# B&R Automation Studio project AP124 (part 3)

#### conveyorP13P14Control.st - not listed in the package file held
```iecst
ACTION ConveyorP13P14Control:

	IF modePalletization = modePalletizationNotReadyToStart THEN
		stateConveyorP13P14 := stateConveyorStop;
	END_IF

	//detect pallet
	IF diPalletStopP14 THEN
		palletOnConveyorP14 := TRUE;
	END_IF

	CASE stateConveyorP13P14 OF

		stateConveyorStop:

			cmdMovePalletP13P14 := FALSE;
			doConveyorP13 := FALSE;
			acpI_P14.switchOn := TRUE;
			acpI_P14.speed := 0;
			acpI_P14.reset := TRUE;
			IF modePalletization <> modePalletizationNotReadyToStart THEN
				stateConveyorP13P14 := stateConveyorWait;
			END_IF

		stateConveyorWait:

			IF cmdMovePalletP13P14 THEN
				IF palletOnConveyorP14 AND NOT diReset THEN
					alarmImagePalletization[3] := TRUE;
					stateConveyorP12P13 := stateConveyorStop;
				ELSE
					TON_ConveyorP13P14(IN := FALSE);
					stateConveyorP13P14 := stateConveyorMoving;
				END_IF
			END_IF

			IF palletOnConveyorP14 > palletOnConveyorP14old THEN
				alarmImagePalletization[10] := TRUE;
				stateConveyorP13P14 := stateConveyorStop;
			END_IF

		stateConveyorMoving:

			doConveyorP13 := TRUE;
			acpI_P14.speed := 500;

			IF NOT cmdMovePalletP13P14 THEN
				stateConveyorP13P14 := stateConveyorStop;
			END_IF

			//sensor reached?
			IF diPalletSlowDownP14 THEN
				palletOnConveyorP13 := FALSE;
				TON_ConveyorP13P14(IN := FALSE);
				stateConveyorP13P14 := stateConveyorMovingSlow;
			END_IF

			//timeout?
			TON_ConveyorP13P14(IN := TRUE, PT := T#12s);
			IF TON_ConveyorP13P14.Q AND NOT diReset THEN
				alarmImagePalletization[4] := TRUE;
				stateConveyorP13P14 := stateConveyorStop;
			END_IF

		stateConveyorMovingSlow:

			acpI_P14.speed := 200;

			IF NOT cmdMovePalletP13P14 THEN
				stateConveyorP13P14 := stateConveyorStop;
			END_IF

			IF palletOnConveyorP14 AND NOT diReset THEN
				stateConveyorP13P14 := stateConveyorStop;
			END_IF

			//timeout?
			TON_ConveyorP13P14(IN := TRUE, PT := T#6s);
			IF TON_ConveyorP13P14.Q AND NOT diReset THEN
				alarmImagePalletization[2] := TRUE;
				stateConveyorP13P14 := stateConveyorStop;
			END_IF
	END_CASE

	//control of ACOPOSinverter P14
	acpI_P14();

	palletOnConveyorP14old := palletOnConveyorP14;

	alarmImagePalletization[13] := NOT diMotorProtectionP13;

	IF acknowledgeImagePalletization[2] THEN
		alarmImagePalletization[2] := FALSE;
	END_IF
	IF acknowledgeImagePalletization[3] THEN
		alarmImagePalletization[3] := FALSE;
	END_IF

	IF acknowledgeImagePalletization[4] THEN
		alarmImagePalletization[4] := FALSE;
	END_IF

	IF acknowledgeImagePalletization[10] THEN
		alarmImagePalletization[10] := FALSE;
	END_IF

	IF acpI_P14.error THEN
		alarmImagePalletization[24] := TRUE;
	ELSE
		alarmImagePalletization[24] := FALSE;
	END_IF

END_ACTION
```

#### conveyorP14.st - not listed in the package file held
```iecst
ACTION ConveyorP14:

	acpI_P14.switchOn := TRUE;
	acpI_P14.speed := 500;

	CASE statePalletP14 OF

		palletNotPresent:

			acpI_P14.run := (cmdMovePalletP14 AND (statePalletP15 = palletNotPresent OR diReset)) OR cmdMovePalletP13;

			//slow down sensor?
			IF diPalletSlowDownP14 THEN
				acpI_P14.speed := 200;
			END_IF

		palletPresent:

			IF cmdMovePalletP14 AND (statePalletP15 = palletNotPresent OR diReset) THEN
				statePalletP14 := palletMoving;
			END_IF

			acpI_P14.run := FALSE;

		palletMoving:

			//sensor reached?
			IF TON_PalletStopP15.Q AND cmdMovePalletP14 AND NOT diReset THEN
				statePalletP15 := palletPresent;
				statePalletP14 := palletNotPresent;
				cmdMovePalletP14 := FALSE;
			END_IF

			acpI_P14.run := cmdMovePalletP14;

	END_CASE

	//control of ACOPOSinverter
	acpI_P14();

END_ACTION
```

#### conveyorP14P15Control.st - not listed in the package file held
```iecst
ACTION ConveyorP14P15Control:

	IF modePalletization = modePalletizationNotReadyToStart THEN
		stateConveyorP14P15 := stateConveyorStop;
	END_IF

	//detect pallet
	IF diPalletStopP15 THEN
		palletOnConveyorP15 := TRUE;
	END_IF

	CASE stateConveyorP14P15 OF

		stateConveyorStop:

			cmdMovePalletP14P15 := FALSE;
			acpI_P14.switchOn := TRUE;
			acpI_P14.speed := 0;
			acpI_P14.reset := TRUE;
			acpI_P15.switchOn := TRUE;
			acpI_P15.speed := 0;
			acpI_P15.reset := TRUE;
			IF modePalletization <> modePalletizationNotReadyToStart THEN
				stateConveyorP14P15 := stateConveyorWait;
			END_IF

		stateConveyorWait:

			IF cmdMovePalletP14P15 THEN
				IF palletOnConveyorP15 AND NOT diReset THEN
					alarmImagePalletization[6] := TRUE;
					stateConveyorP14P15 := stateConveyorStop;
				ELSE
					TON_ConveyorP14P15(IN := FALSE);
					stateConveyorP14P15 := stateConveyorMoving;
				END_IF
			END_IF

			IF palletOnConveyorP15 > palletOnConveyorP15old THEN
				alarmImagePalletization[11] := TRUE;
				stateConveyorP14P15 := stateConveyorStop;
			END_IF

		stateConveyorMoving:

			acpI_P14.speed := 500;
			acpI_P15.speed := 500;

			IF NOT cmdMovePalletP14P15 THEN
				stateConveyorP14P15 := stateConveyorStop;
			END_IF

			//sensor reached?
			IF palletOnConveyorP15 AND NOT diReset THEN
				palletOnConveyorP14 := FALSE;
				stateConveyorP14P15 := stateConveyorStop;
			END_IF

			//timeout?
			TON_ConveyorP14P15(IN := TRUE, PT := T#12s);
			IF TON_ConveyorP14P15.Q AND NOT diReset THEN
				alarmImagePalletization[7] := TRUE;
				stateConveyorP14P15 := stateConveyorStop;
			END_IF

	END_CASE

	//control of ACOPOSinverter P15
	acpI_P15();

	palletOnConveyorP15old := palletOnConveyorP15;

	IF acknowledgeImagePalletization[6] THEN
		alarmImagePalletization[6] := FALSE;
	END_IF
	IF acknowledgeImagePalletization[7] THEN
		alarmImagePalletization[7] := FALSE;
	END_IF

	IF acknowledgeImagePalletization[11] THEN
		alarmImagePalletization[11] := FALSE;
	END_IF

	IF acpI_P15.error THEN
		alarmImagePalletization[25] := TRUE;
	ELSE
		alarmImagePalletization[25] := FALSE;
	END_IF

END_ACTION
```

#### conveyorP15.st - not listed in the package file held
```iecst
ACTION ConveyorP15:

	acpI_P15.switchOn := TRUE;
	acpI_P15.speed := 500;

	CASE statePalletP15 OF

		palletNotPresent:

			acpI_P15.run := (cmdMovePalletP15 AND (statePalletP16 = palletNotPresent OR diReset)) OR cmdMovePalletP14;

		palletPresent:

			IF cmdMovePalletP15 AND (statePalletP16 = palletNotPresent OR diReset) THEN
				statePalletP15 := palletMoving;
			END_IF

			acpI_P15.run := FALSE;

		palletMoving:

			//sensor reached?
			IF TON_PalletStopP16.Q AND cmdMovePalletP15 AND NOT diReset THEN
				statePalletP16 := palletPresent;
				statePalletP15 := palletNotPresent;
				cmdMovePalletP15 := FALSE;
			END_IF

			acpI_P15.run := cmdMovePalletP15;

	END_CASE

	//control of ACOPOSinverter
	acpI_P15();

END_ACTION
```

#### conveyorP16.st - not listed in the package file held
```iecst
ACTION ConveyorP16:

	acpI_P16.switchOn := TRUE;
	acpI_P16.speed := 500;

	CASE statePalletP16 OF

		palletNotPresent:

			acpI_P16.run := (cmdMovePalletP16 AND (statePalletP17 = palletNotPresent OR diReset)) OR cmdMovePalletP15;

		palletPresent:

			IF cmdMovePalletP16 AND (statePalletP17 = palletNotPresent OR diReset) THEN
				statePalletP16 := palletMoving;
			END_IF

			acpI_P16.run := FALSE;

		palletMoving:

			//sensor reached?
			IF TON_PalletStopP17.Q AND cmdMovePalletP16 AND NOT diReset THEN
				statePalletP17 := palletPresent;
				statePalletP16 := palletNotPresent;
				cmdMovePalletP16 := FALSE;
			END_IF

			acpI_P16.run := cmdMovePalletP16;

	END_CASE

	//control of ACOPOSinverter
	acpI_P16();

END_ACTION
```

#### conveyorP17.st - not listed in the package file held
```iecst
ACTION ConveyorP17:

	acpI_P17.switchOn := TRUE;
	acpI_P17.speed := 500;

	CASE statePalletP17 OF

		palletNotPresent:

			acpI_P17.run := (cmdMovePalletP17 AND (statePalletP18 = palletNotPresent OR diReset) AND stateTurnTable = stateTurnTableEntryPosition) OR cmdMovePalletP16;

		palletPresent:

			IF cmdMovePalletP17 AND (statePalletP18 = palletNotPresent OR diReset) THEN
				statePalletP17 := palletMoving;
			END_IF

			acpI_P17.run := FALSE;

		palletMoving:

			//sensor reached?
			IF TON_PalletStopP18.Q AND cmdMovePalletP17 AND NOT diReset THEN
				statePalletP18 := palletPresent;
				statePalletP17 := palletNotPresent;
				cmdMovePalletP17 := FALSE;
			END_IF

			acpI_P17.run := cmdMovePalletP17;

	END_CASE

	//control of ACOPOSinverter
	acpI_P17();

END_ACTION
```

### pallet_conveyors.typ - not listed in the package file held
```iecst
TYPE
	ModeConveyors :
		(
		modeConveyorsNotReadyToStart,
		modeConveyorsManual,
		modeConveyorsAuto
		);
END_TYPE
```

### outfeed.typ
```iecst
TYPE
	StateTurnTable :
		(
		stateTurnTableInit,
		stateTurnTableEntryPosition,
		stateTurnTableMovingToExitPos,
		stateTurnTableExitPosition,
		stateTurnTableMovingToEntryPos
		);
END_TYPE
```

### outfeed.var
```iecst
VAR
	acknowledgeImageOutfeed : ARRAY[0..39] OF BOOL;
	alarmImageOutfeed : ARRAY[0..39] OF BOOL;
	alarmInZoneOutfeed : BOOL;
	cmdMovePalletP17 : BOOL;
	cmdMovePalletP18 : BOOL;
	cmdOutfeedAuto : BOOL; (*VISU:switches pallet magazine to automatic mode*)
	cmdOutfeedManual : BOOL;
	diWrapperDoorCanBeOpened : BOOL;
	diWrapperEntryFree : BOOL;
	diWrapperExitFree : BOOL;
	diWrapperInAuto : BOOL;
	diWrapperLowFoil : BOOL;
	diWrapperNoError : BOOL;
	diWrappingFinished : BOOL;
	doWrapperNoExternalStop : BOOL;
	doWrapperSortiment1 : BOOL;
	doWrapperSortiment2 : BOOL;
	doWrappingStart : BOOL;
	modeZoneOutfeed : ModeZone;
	modeZoneOutfeedOld : ModeZone;
	statePalletP17 : StatePallet;
	statePalletP18 : StatePallet;
	statePalletP19 : StatePallet;
	statePalletP20 : StatePallet;
	statePalletP21 : StatePallet;
	statePalletP22 : StatePallet;
	stateTurnTable : StateTurnTable;
END_VAR
```

### Program Logical/plc/outfeed/outfeed_main (IEC) - palletization state machine

#### outfeed_main.st - Init, cyclic, exit code
```iecst
PROGRAM _INIT

END_PROGRAM

PROGRAM _CYCLIC

	modeZoneOutfeedOld := modeZoneOutfeed;

	readyToStart := NOT diOutfeedEDM;

	IF cpuIsSimulated THEN
		readyToStart := TRUE;
	END_IF

	IF NOT readyToStart THEN
		modeZoneOutfeed := modeZoneOff;
	END_IF

	CASE modeZoneOutfeed OF

		modeZoneOff: //the automat is not ready to start

			cmdOutfeedManual := FALSE;
			cmdOutfeedAuto := FALSE;

			IF readyToStart THEN
				modeZoneOutfeed := modeZoneManual;
			END_IF

		modeZoneManual:

			cmdOutfeedManual := FALSE;

			IF (NOT alarmInZoneOutfeed OR cpuIsSimulated) AND cmdOutfeedAuto THEN
				modeZoneOutfeed := modeZoneAuto;
			END_IF

		modeZoneAuto:

			cmdOutfeedAuto := FALSE;

			IF (alarmInZoneOutfeed AND NOT cpuIsSimulated) OR cmdOutfeedManual THEN
				modeZoneOutfeed := modeZoneManual;
			END_IF

	END_CASE

	//alarms
	alarmImageOutfeed[0] := NOT lightCurtainP17;
	alarmImageOutfeed[3] := NOT diMotorProtectionP19;
	alarmImageOutfeed[9] := NOT diMotorProtectionP20;
	alarmImageOutfeed[12] := NOT diMotorProtectionP21;
	alarmImageOutfeed[13] := NOT diMotorProtectionP22;
END_PROGRAM
```

#### outfeed_main.var - Local variables
```iecst
VAR
	readyToStart : BOOL;
	diMotorProtectionP19 : BOOL;
	diMotorProtectionP20 : BOOL;
	diMotorProtectionP21 : BOOL;
	diMotorProtectionP22 : BOOL;
	lightCurtainP17 : BOOL;
END_VAR
```

### Program Logical/plc/outfeed/pallet_outfeed/pallet_outfeed (IEC) - pallet outfeed control

#### Main.st - Cyclic code
```iecst
PROGRAM _INIT
	(* Insert code here *)

END_PROGRAM

PROGRAM _CYCLIC
	TON_PalletStopP18(IN := diPalletStopP18, PT := T#200ms);
	TON_PalletStopP20(IN := diPalletStopP20, PT := T#200ms);
	TON_PalletStopP21(IN := diPalletStopP21, PT := T#200ms);
	TON_PalletStopP22(IN := diPalletStopP22, PT := T#200ms);

	CASE modeZoneOutfeed OF

		modeZoneOff:

		modeZoneManual:

			IF modeZoneOutfeedOld <> modeZoneManual THEN
				cmdMovePalletP17 := FALSE;
				cmdMovePalletP19 := FALSE;
				cmdMovePalletP20 := FALSE;
				cmdMovePalletP21 := FALSE;
				cmdMovePalletP22 := FALSE;
			END_IF

		modeZoneAuto:

			//stop sensor not reached
			TON_ConveyorP17(IN := cmdMovePalletP17, PT := T#20s);
			alarmImageOutfeed[21] := TON_ConveyorP17.Q;

			TON_ConveyorP19(IN := cmdMovePalletP19, PT := T#20s);
			alarmImageOutfeed[1] := TON_ConveyorP19.Q;

			TON_ConveyorP20(IN := cmdMovePalletP20, PT := T#20s);
			alarmImageOutfeed[8] := TON_ConveyorP20.Q;

			TON_ConveyorP21(IN := cmdMovePalletP21, PT := T#20s);
			alarmImageOutfeed[11] := TON_ConveyorP21.Q;

			// control conveyors
			IF statePalletP17 <> palletNotPresent AND statePalletP18 = palletNotPresent AND stateTurnTable = stateTurnTableEntryPosition AND diWrapperEntryFree THEN
				cmdMovePalletP17 := TRUE;
			END_IF

			IF statePalletP19 <> palletNotPresent AND statePalletP20 = palletNotPresent THEN
				cmdMovePalletP19 := TRUE;
			END_IF

			IF statePalletP20 <> palletNotPresent AND statePalletP21 = palletNotPresent THEN
				cmdMovePalletP20 := TRUE;
			END_IF

			IF statePalletP21 <> palletNotPresent AND statePalletP22 = palletNotPresent THEN
				cmdMovePalletP21 := TRUE;
			END_IF

			//unexpected pallet
			IF TON_PalletStopP18.Q AND statePalletP18 = palletNotPresent AND NOT cmdMovePalletP17 AND stateTurnTable = stateTurnTableEntryPosition THEN
				alarmImageOutfeed[20] := TRUE;
			END_IF
			IF TON_PalletStopP20.Q AND statePalletP20 = palletNotPresent AND NOT cmdMovePalletP19 THEN
				alarmImageOutfeed[2] := TRUE;
			END_IF
			IF TON_PalletStopP21.Q AND statePalletP21 = palletNotPresent AND NOT cmdMovePalletP20 THEN
				alarmImageOutfeed[7] := TRUE;
			END_IF
			IF TON_PalletStopP22.Q AND statePalletP22 = palletNotPresent AND NOT cmdMovePalletP21 THEN
				alarmImageOutfeed[10] := TRUE;
			END_IF

	END_CASE

	//conveyors
	ConveyorP17;
	ConveyorP19;
	ConveyorP20;
	ConveyorP21;
	ConveyorP22;

	//stop sensor not reached
	IF acknowledgeImageOutfeed[21] THEN
		alarmImageOutfeed[21] := FALSE;
	END_IF
	IF acknowledgeImageOutfeed[1] THEN
		alarmImageOutfeed[1] := FALSE;
	END_IF
	IF acknowledgeImageOutfeed[8] THEN
		alarmImageOutfeed[8] := FALSE;
	END_IF
	IF acknowledgeImageOutfeed[11] THEN
		alarmImageOutfeed[11] := FALSE;
	END_IF

	//unexpected pallet
	IF acknowledgeImageOutfeed[20] THEN
		alarmImageOutfeed[20] := FALSE;
	END_IF
	IF acknowledgeImageOutfeed[2] THEN
		alarmImageOutfeed[2] := FALSE;
	END_IF
	IF acknowledgeImageOutfeed[7] THEN
		alarmImageOutfeed[7] := FALSE;
	END_IF
	IF acknowledgeImageOutfeed[10] THEN
		alarmImageOutfeed[10] := FALSE;
	END_IF

	//problems with motors
	acknowledgeImageOutfeed[22] := acpI_P17.error;
	acpI_P17.reset := EDGENEG(acknowledgeImageOutfeed[22]);

END_PROGRAM
```

#### Variables.var - Local variables
```iecst
VAR
	acpI_P17 : AcpInoSdc;
	cmdMovePalletP19 : BOOL;
	cmdMovePalletP20 : BOOL;
	cmdMovePalletP21 : BOOL;
	cmdMovePalletP22 : BOOL;
	diPalletStopP18 : BOOL;
	diPalletStopP20 : BOOL;
	diPalletStopP21 : BOOL;
	diPalletStopP22 : BOOL;
	doConveyorP19 : BOOL;
	doConveyorP20 : BOOL;
	doConveyorP21 : BOOL;
	doConveyorP22 : BOOL;
	TOF_PalletStopP22 : TOF;
	TON_ConveyorP17 : TON;
	TON_ConveyorP19 : TON;
	TON_ConveyorP20 : TON;
	TON_ConveyorP21 : TON;
	TON_PalletStopP18 : TON;
	TON_PalletStopP20 : TON;
	TON_PalletStopP21 : TON;
	TON_PalletStopP22 : TON;
END_VAR
```

#### conveyorP19.st
```iecst
ACTION ConveyorP19:

	CASE statePalletP19 OF

		palletNotPresent:

			doConveyorP19 := (cmdMovePalletP19 AND (statePalletP20 = palletNotPresent OR diReset)) OR (cmdMovePalletP18 AND stateTurnTable = stateTurnTableExitPosition);

		palletPresent:

			IF cmdMovePalletP19 AND (statePalletP20 = palletNotPresent OR diReset) THEN
				statePalletP19 := palletMoving;
			END_IF

			doConveyorP19 := FALSE;

		palletMoving:

			//sensor reached?
			IF TON_PalletStopP20.Q AND cmdMovePalletP19 AND NOT diReset THEN
				statePalletP20 := palletPresent;
				statePalletP19 := palletNotPresent;
				cmdMovePalletP19 := FALSE;
			END_IF

			doConveyorP19 := cmdMovePalletP19;

	END_CASE

END_ACTION
```

#### conveyorP20.st
```iecst
ACTION ConveyorP20:

	CASE statePalletP20 OF

		palletNotPresent:

			doConveyorP20 := (cmdMovePalletP20 AND (statePalletP21 = palletNotPresent OR diReset)) OR cmdMovePalletP19;

		palletPresent:

			IF cmdMovePalletP20 AND (statePalletP21 = palletNotPresent OR diReset) THEN
				statePalletP20 := palletMoving;
			END_IF

			doConveyorP20 := FALSE;

		palletMoving:

			//sensor reached?
			IF TON_PalletStopP21.Q AND cmdMovePalletP20 AND NOT diReset THEN
				statePalletP21 := palletPresent;
				statePalletP20 := palletNotPresent;
				cmdMovePalletP20 := FALSE;
			END_IF

			doConveyorP20 := cmdMovePalletP20;

	END_CASE

END_ACTION
```

#### conveyorP21.st
```iecst
ACTION ConveyorP21:

	CASE statePalletP21 OF

		palletNotPresent:

			doConveyorP21 := (cmdMovePalletP21 AND (statePalletP22 = palletNotPresent OR diReset)) OR cmdMovePalletP20;

		palletPresent:

			IF cmdMovePalletP21 AND (statePalletP22 = palletNotPresent OR diReset) THEN
				statePalletP21 := palletMoving;
			END_IF

			doConveyorP21 := FALSE;

		palletMoving:

			//sensor reached?
			IF TON_PalletStopP22.Q AND cmdMovePalletP21 AND NOT diReset THEN
				statePalletP22 := palletPresent;
				statePalletP21 := palletNotPresent;
				cmdMovePalletP21 := FALSE;
			END_IF

			doConveyorP21 := cmdMovePalletP21;

	END_CASE

END_ACTION
```

#### conveyorP22.st
```iecst
ACTION ConveyorP22:

	TOF_PalletStopP22(IN := diPalletStopP22, PT := T#30s);

	IF NOT TOF_PalletStopP22.Q THEN
		statePalletP22 := palletNotPresent;
	END_IF

	CASE statePalletP22 OF

		palletNotPresent:

			doConveyorP22 := (cmdMovePalletP22 AND diReset) OR cmdMovePalletP21;

		palletPresent:

			doConveyorP22 := FALSE;

		palletMoving:

			statePalletP22 := palletNotPresent;

	END_CASE

END_ACTION
```

### Program Logical/plc/outfeed/wrapper/wrapper (IEC)

#### Main.st - Cyclic code
```iecst
PROGRAM _INIT

	diWrapperDoorCanBeOpened;

END_PROGRAM

PROGRAM _CYCLIC

	IF adrRecipes = 0 THEN
		RETURN;
	END_IF

	dRecipes ACCESS adrRecipes;
	IF dRecipes.actualRecipeIndex < 0 OR dRecipes.actualRecipeIndex > 9 THEN
		RETURN;
	END_IF

	dActualRecipe ACCESS ADR(dRecipes.recipe[dRecipes.actualRecipeIndex]);

	doWrapperSortiment1 := dActualRecipe.wrapperSortiment.0;
	doWrapperSortiment2 := dActualRecipe.wrapperSortiment.1;

	IF testAtAtrima THEN
		diPalletStopP19 := FALSE;
	END_IF

	TON_PalletStopP19(IN := diPalletStopP19, PT := T#200ms);

	CASE modeZoneOutfeed OF

		modeZoneOff: //the automat is not ready to start

		modeZoneManual:

			IF modeZoneOutfeedOld <> modeZoneManual THEN
				cmdMovePalletP18 := FALSE;
			END_IF

			doWrapperNoExternalStop := TRUE;
			doWrappingStart := FALSE;
			stateAuto := stateAutoUndefined;

		modeZoneAuto:

			//stop sensor not reached
			TON_ConveyorP18(IN := cmdMovePalletP18, PT := T#20s);
			alarmImageOutfeed[4] := TON_ConveyorP18.Q;

			CASE stateAuto OF

				stateAutoUndefined:

					IF stateTurnTable = stateTurnTableEntryPosition THEN
						stateAuto := stateAutoWait;
					ELSE
						stateAuto := stateAutoRemovePallet;
					END_IF

				stateAutoWait:

					IF statePalletP18 = palletPresent AND stateTurnTable = stateTurnTableEntryPosition AND diWrapperInAuto THEN
						TON_Wrapper(IN:=FALSE);
						stateAuto := stateAutoWait2;
					END_IF

				stateAutoWait2:

					TON_Wrapper(IN:=TRUE, PT:=T#2s);
					IF TON_Wrapper.Q THEN
						stateAuto := stateAutoRun;
					END_IF

				stateAutoRun:

					doWrappingStart := TRUE;

					IF diWrappingFinished THEN
						stateAuto := stateAutoTurnToExitPosition;
					END_IF

				stateAutoTurnToExitPosition:

					doWrappingStart := FALSE;
					cmdTurnToExitPosition := TRUE;
					stateAuto := stateAutoWaitForExitPosition;

				stateAutoWaitForExitPosition:

					IF stateTurnTable = stateTurnTableExitPosition THEN
						stateAuto := stateAutoRemovePallet;
					END_IF

				stateAutoRemovePallet:

					IF statePalletP18 <> palletNotPresent AND statePalletP19 = palletNotPresent AND stateTurnTable = stateTurnTableExitPosition AND diWrapperExitFree THEN
						cmdMovePalletP18 := TRUE;
					END_IF

					IF statePalletP18 = palletNotPresent THEN
						stateAuto := stateAutoTurnToEntryPosition;
					END_IF

				stateAutoTurnToEntryPosition:

					cmdTurnToEntryPosition := TRUE;
					stateAuto := stateAutoWaitForEntryPosition;

				stateAutoWaitForEntryPosition:

					IF stateTurnTable = stateTurnTableEntryPosition THEN
						stateAuto := stateAutoWait;
					END_IF

			END_CASE

			//unexpected pallet
			IF TON_PalletStopP19.Q AND statePalletP19 = palletNotPresent AND NOT cmdMovePalletP18 THEN
				alarmImageOutfeed[5] := TRUE;
			END_IF
	END_CASE

	//modules
	ConveyorP18;
	TurnTable;

	//door logic
	DoorLogic_2();
	alarmImageOutfeed[15] := NOT DoorLogic_2.diDoorLocked;

	alarmImageOutfeed[16] := wrapperEdmError;
	alarmImageOutfeed[17] := NOT diWrapperNoError;
	alarmImageOutfeed[18] := diWrapperLowFoil;
	alarmImageOutfeed[19] := NOT diWrapperInAuto;

	//sensor not reached
	IF acknowledgeImageOutfeed[4] THEN
		alarmImageOutfeed[4] := FALSE;
	END_IF

	//unexpected pallet
	IF acknowledgeImageOutfeed[5] THEN
		alarmImageOutfeed[5] := FALSE;
	END_IF

	//problems with motors
	alarmImageOutfeed[6] := acpI_P18_1.error;
	acpI_P18_1.reset := EDGENEG(acknowledgeImageOutfeed[6]);

	alarmImageOutfeed[14] := acpI_P18_2.error;
	acpI_P18_2.reset := EDGENEG(acknowledgeImageOutfeed[14]);

END_PROGRAM
```

#### Types.typ - Local data types
```iecst
TYPE
	StateAuto :
		(
		stateAutoUndefined,
		stateAutoWait,
		stateAutoWait2,
		stateAutoRun,
		stateAutoTurnToExitPosition,
		stateAutoWaitForExitPosition,
		stateAutoRemovePallet,
		stateAutoTurnToEntryPosition,
		stateAutoWaitForEntryPosition
		);
END_TYPE
```

#### Variables.var - Local variables
```iecst
VAR
	acpI_P18_1 : AcpInoSdc;
	acpI_P18_2 : AcpInoSdc;
	cmdTurnToEntryPosition : BOOL;
	cmdTurnToExitPosition : BOOL;
	conveyorP18speed : INT;
	diEntrySwitch : BOOL;
	diExitSwitch : BOOL;
	diPalletStopP19 : BOOL;
	DoorLogic_2 : DoorLogic;
	TON_ConveyorP18 : TON;
	TON_PalletStopP19 : TON;
	turnTableSpeed : INT;
	wrapperEdmError : BOOL;
	stateAuto : StateAuto;
	dRecipes : REFERENCE TO Recipes;
	dActualRecipe : REFERENCE TO Recipe;
	TON_Wrapper : TON;
END_VAR
```

#### conveyorP18.st
```iecst
ACTION ConveyorP18:

	acpI_P18_1.switchOn := TRUE;
	conveyorP18speed := 635;//500;

	IF stateTurnTable = stateTurnTableEntryPosition THEN
		acpI_P18_1.speed := conveyorP18speed;
	END_IF

	IF stateTurnTable = stateTurnTableExitPosition THEN
		acpI_P18_1.speed := -conveyorP18speed;
	END_IF

	CASE statePalletP18 OF

		palletNotPresent:

			acpI_P18_1.run := (cmdMovePalletP18 AND (statePalletP18 = palletNotPresent OR diReset)) OR (cmdMovePalletP17 AND stateTurnTable = stateTurnTableEntryPosition);

		palletPresent:

			IF cmdMovePalletP18 AND (statePalletP19 = palletNotPresent OR diReset) THEN
				statePalletP18 := palletMoving;
			END_IF

			acpI_P18_1.run := FALSE;

		palletMoving:

			//sensor reached?
			IF TON_PalletStopP19.Q AND cmdMovePalletP18 AND NOT diReset THEN
				statePalletP19 := palletPresent;
				statePalletP18 := palletNotPresent;
				cmdMovePalletP18 := FALSE;
			END_IF

			acpI_P18_1.run := cmdMovePalletP18 AND (stateTurnTable = stateTurnTableExitPosition);

	END_CASE

	//lock movement
	IF stateTurnTable <> stateTurnTableEntryPosition AND stateTurnTable <> stateTurnTableExitPosition THEN
		acpI_P18_1.run := FALSE;
	END_IF

	//control of ACOPOSinverter
	acpI_P18_1();

END_ACTION
```

#### turnTable.st
```iecst
ACTION TurnTable:

	acpI_P18_2.switchOn := TRUE;
	turnTableSpeed := 1500;

	CASE stateTurnTable OF

		stateTurnTableInit:

			acpI_P18_2.run := FALSE;

			IF diEntrySwitch THEN
				stateTurnTable := stateTurnTableEntryPosition;
			END_IF

			IF diExitSwitch THEN
				stateTurnTable := stateTurnTableExitPosition;
			END_IF

			IF stateTurnTable = stateTurnTableInit THEN

				IF cmdTurnToEntryPosition THEN
					stateTurnTable := stateTurnTableMovingToEntryPos;
				END_IF

				IF cmdTurnToExitPosition THEN
					stateTurnTable := stateTurnTableMovingToExitPos;
				END_IF
			END_IF

		stateTurnTableEntryPosition:

			IF cmdTurnToExitPosition THEN
				stateTurnTable := stateTurnTableMovingToExitPos;
			END_IF

			cmdTurnToEntryPosition := FALSE;

		stateTurnTableMovingToExitPos:

			acpI_P18_2.speed := turnTableSpeed;
			acpI_P18_2.run := TRUE;

			IF diExitSwitch OR NOT cmdTurnToExitPosition THEN
				StopMovement;
			END_IF

		stateTurnTableExitPosition:

			IF cmdTurnToEntryPosition THEN
				stateTurnTable := stateTurnTableMovingToEntryPos;
			END_IF

			cmdTurnToExitPosition := FALSE;

		stateTurnTableMovingToEntryPos:

			acpI_P18_2.speed := -turnTableSpeed;
			acpI_P18_2.run := TRUE;

			IF diEntrySwitch OR NOT cmdTurnToEntryPosition THEN
				StopMovement;
			END_IF

	END_CASE

	//control of ACOPOSinverter
	acpI_P18_2();

END_ACTION

ACTION StopMovement:
	cmdTurnToEntryPosition := FALSE;
	cmdTurnToExitPosition := FALSE;
	stateTurnTable := stateTurnTableInit;
END_ACTION
```

### alarm_management.var
```iecst
VAR
	alarmCommon : BOOL;
	alarmImageCommon : ARRAY[0..39] OF BOOL;
	alarmInZoneMagazine : BOOL; (*VISU:there is at least one alarm in pallet magazine*)
	cpuIsSimulated : BOOL;
	diAirPresureOK : BOOL; (*VISU: 1...air pressure OK*)
	diReset : BOOL; (*acknowledges all errors*)
	alarmPresent : BOOL;
	safetyAlive : BOOL;
END_VAR
```

### Program Logical/plc/alarm_management/alarm_management (IEC) - alarm management

#### Variables.var
```iecst
VAR
	acknowledgeImage : ARRAY[0..39] OF BOOL;
	diEStop1 : BOOL; (*emergency stop 1*)
	diEStop2 : BOOL; (*emergency stop 2*)
	diEStop3 : BOOL; (*emergency stop 3*)
	diEStop4 : BOOL; (*emergency stop 4*)
	diEStopRobot : BOOL; (*emergency stop - robot*)
	diEStopWrapper : BOOL; (*emergency stop wrapper*)
	i : INT;
	magazineEdmError : BOOL; (*1=power on*)
	outfeedEdmError : BOOL; (*1=power on*)
	palletizationEdmError : BOOL; (*1=power on*)
	diEStop5 : BOOL;
END_VAR
```

#### Cyclic.st
```iecst
PROGRAM _CYCLIC

	MpAlarmXCore_0.MpLink := ADR(gAlarmXCore);
	MpAlarmXCore_0.Enable := 1;

	MpAlarmXCore_0();

	MpAlarmXListUI_0.MpLink := ADR(gAlarmXCore);
	MpAlarmXListUI_0.Enable := 1;
	MpAlarmXListUI_0.UIConnect := ADR(MpAlarmXListUIConnect);
	MpAlarmXListUI_0();

	IF diAirPresureOK THEN
		MpAlarmXReset(gAlarmXCore,'AirPressureNotOK');
	ELSE
		MpAlarmXSet(gAlarmXCore,'AirPressureNotOK');
	END_IF

	IF EDGEPOS(diReset) THEN
		MpAlarmXListUIConnect.AcknowledgeAll := TRUE;
	END_IF

END_PROGRAM
```

#### Main.st
```iecst
PROGRAM _INIT

	cpuIsSimulated := DiagCpuIsSimulated();

END_PROGRAM

PROGRAM _CYCLIC

	alarmImageCommon[0] := NOT diAirPresureOK;
	alarmImageCommon[1] := NOT diEStop1;
	alarmImageCommon[2] := NOT diEStop2;
	alarmImageCommon[3] := NOT diEStop3;
	alarmImageCommon[4] := NOT diEStop4;
	alarmImageCommon[14] := NOT diEStop5;

	alarmImageCommon[5] := NOT diEStopRobot;
	alarmImageCommon[6] := NOT diEStopWrapper;
	alarmImageCommon[7] := NOT safetyAlive;

	alarmImageCommon[8] := diMagazineEDM;
	alarmImageCommon[9] := diPalletizationEDM;
	alarmImageCommon[10] := diOutfeedEDM;
	alarmImageCommon[11] := magazineEdmError;
	alarmImageCommon[12] := palletizationEdmError;
	alarmImageCommon[13] := outfeedEdmError;

	//detect if there is any alarm
	alarmCommon := FALSE;
	FOR i:=0 TO 39 DO
		IF alarmImageCommon[i] OR acknowledgeImage[i] THEN
			alarmCommon := TRUE;
		END_IF
	END_FOR

	//detect if there is any alarm in zone Magazine
	alarmInZoneMagazine := FALSE;
	FOR i:=0 TO 39 DO
		IF alarmImageMagazine[i] OR acknowledgeImageMagazine[i] THEN
			alarmInZoneMagazine := TRUE;
		END_IF
	END_FOR

	//detect if there is any alarm in zone Palletization
	alarmInZonePalletization := FALSE;
	FOR i:=0 TO 69 DO
		IF alarmImagePalletization[i] OR acknowledgeImagePalletization[i] THEN
			alarmInZonePalletization := TRUE;
		END_IF
	END_FOR

	//detect if there is any alarm in zone Outfeed
	alarmInZoneOutfeed := FALSE;
	FOR i:=0 TO 39 DO
		IF alarmImageOutfeed[i] OR acknowledgeImageOutfeed[i] THEN
			alarmInZoneOutfeed := TRUE;
		END_IF
	END_FOR

	IF alarmCommon OR alarmInZoneMagazine OR alarmInZonePalletization OR alarmInZoneOutfeed THEN
		alarmPresent := TRUE;
	ELSE
		alarmPresent := FALSE;
	END_IF

END_PROGRAM
```

### recipe_management.typ
```iecst
TYPE
	Layout : 	STRUCT
		nbOfTrays : INT;
		tray : ARRAY[0..39]OF Tray;
	END_STRUCT;
	Recipe : 	STRUCT
		name : STRING[80];
		interlayerSheetBottom : BOOL;
		interlayerSheetTop : BOOL;
		conveyorP1speed : INT;
		conveyorP2speed : INT;
		timeAfterLastTrayInRow : TIME;
		timeDelayForTurn : TIME;
		nbOfLayers : INT;
		layer : ARRAY[0..9]OF INT;
	END_STRUCT;
	Recipes : 	STRUCT
		actualRecipeIndex : INT;
		recipe : ARRAY[0..9]OF Recipe;
		layout : ARRAY[0..9]OF Layout;
	END_STRUCT;
	Tray : 	STRUCT
		turnTray : BOOL;
		lastTray : LastTray;
	END_STRUCT;
	LastTray :
		(
		lastTrayNo,
		lastTrayInRow,
		lastTrayInHalfLayer,
		lastTrayInLayer
		);
END_TYPE
```

### recipe_management.var
```iecst
VAR
	adrRecipes : UDINT;
END_VAR
```

### Program Logical/plc/recipe_management/recipe_management (IEC)

#### Types.typ
```iecst
TYPE
	StateRecipe :
		(
		stateRecipeError,
		stateRecipeInit,
		stateRecipeWait,
		stateRecipeLoad,
		stateRecipeLoad2,
		stateRecipeLoad3,
		stateRecipeSave,
		stateRecipeSave2,
		stateRecipeSave3
		);
END_TYPE
```

#### Variables.var
```iecst
VAR
	cmdLoad : BOOL;
	cmdSave : BOOL;
	MpRecipeCsv_0 : MpRecipeCsv;
	MpRecipeRegPar_0 : MpRecipeRegPar;
	readyToStart : BOOL;
	recipes : Recipes;
	stateRecipe : StateRecipe;
END_VAR
```

#### Main.st
```iecst
PROGRAM _INIT

END_PROGRAM

PROGRAM _CYCLIC

	adrRecipes := ADR(recipes);

	readyToStart :=  NOT MpRecipeRegPar_0.Error AND NOT MpRecipeCsv_0.Error;

	IF NOT readyToStart THEN
		stateRecipe := stateRecipeError;
	END_IF

	CASE stateRecipe OF

		stateRecipeError:

			cmdLoad := FALSE;
			cmdSave := FALSE;
			VisuRecipeState := 4;							//Visu Error Text
			IF readyToStart THEN
				stateRecipe := stateRecipeInit;
			END_IF

		stateRecipeInit:

			MpRecipeRegPar_0.MpLink := ADR(gRecipeCsv);
			MpRecipeRegPar_0.Enable := TRUE;
			MpRecipeRegPar_0.PVName := ADR('recipe_man:recipes');

			MpRecipeCsv_0.MpLink := ADR(gRecipeCsv);
			MpRecipeCsv_0.Enable := TRUE;
			MpRecipeCsv_0.DeviceName := ADR('USER');
			MpRecipeCsv_0.FileName := ADR('recipe.csv');

			VisuRecipeState := 0;						//Visu Empty Text

			IF MpRecipeRegPar_0.Active AND MpRecipeCsv_0.Active THEN
				stateRecipe := stateRecipeLoad;
			END_IF

		stateRecipeWait:

			IF cmdLoad THEN
				stateRecipe := stateRecipeLoad;
			END_IF

			IF cmdSave THEN
				stateRecipe := stateRecipeSave;
			END_IF

		stateRecipeLoad:

			MpRecipeCsv_0.Load := TRUE;
			stateRecipe := stateRecipeLoad2;
			VisuRecipeState := 3;						//Visu Discart changes Text

		stateRecipeLoad2:

			IF MpRecipeCsv_0.CommandDone THEN
				cmdLoad := FALSE;
				MpRecipeCsv_0.Load := FALSE;
				stateRecipe := stateRecipeWait;
				VisuRecipeState := 0;					//Visu Empty Text
				RecipeChanged := TRUE;
			END_IF

		stateRecipeSave:

			MpRecipeCsv_0.Save := TRUE;
			stateRecipe := stateRecipeSave2;
			VisuRecipeState := 1;						//Visu Saving Text

		stateRecipeSave2:

			IF MpRecipeCsv_0.CommandDone THEN
				cmdSave := FALSE;
				MpRecipeCsv_0.Save := FALSE;
				stateRecipe := stateRecipeWait;
				VisuRecipeState := 2;					//Visu Saved Text
				RecipeChanged := TRUE;
			END_IF

	END_CASE

	MpRecipeRegPar_0();
	MpRecipeCsv_0();

END_PROGRAM

PROGRAM _EXIT
	MpRecipeRegPar_0(Enable := FALSE);
	MpRecipeCsv_0(Enable := FALSE);
END_PROGRAM
```

### misc.var
```iecst
VAR
	testAtAtrima : BOOL;
	diActivateAllSafetyCircuits : BOOL; (*button on main cabinet to activate all safety circuits*)
	diMagazineEDM : BOOL; (*magazine safety zone: 0...contactor switched on*)
	diPalletizationEDM : BOOL; (*paletization safety zone: 0...contactor switched on*)
	diOutfeedEDM : BOOL; (*wrapper+outfeed safety zone: 0...contactor switched on*)
END_VAR
```

### Program Logical/plc/misc/misc

#### Variables.var
```iecst
VAR
	doLedOn : BOOL; (*LED indicator on main cabinet*)
	doLedOff : BOOL; (*LED indicator on main cabinet*)
	MTBasicsPWM_2 : MTBasicsPWM;
	MTBasicsPWM_1 : MTBasicsPWM;
	MTBasicsPWM_0 : MTBasicsPWM;
	sumEDM : INT;
	doSafetyCurtainSupplyP15 : BOOL;
	doSafetyCurtainSupplyP17 : BOOL;
	doSafetyCurtainSupplyP11 : BOOL;
	doSignColumnGreen : BOOL;
	doSignColumnOrange : BOOL;
	doSignColumnRed : BOOL;
	doSignColumnHorn : BOOL;
	sumAuto : INT;
	bypassHorn : BOOL;
END_VAR
```

#### Main.st
```iecst
PROGRAM _INIT

	doSafetyCurtainSupplyP11 := TRUE;
	doSafetyCurtainSupplyP15 := TRUE;
	doSafetyCurtainSupplyP17 := TRUE;

END_PROGRAM

PROGRAM _CYCLIC

	sumEDM := BOOL_TO_INT(diMagazineEDM) + BOOL_TO_INT(diPalletizationEDM) + BOOL_TO_INT(diOutfeedEDM);

	CASE sumEDM OF
		0:
			MTBasicsPWM_0.DutyCycle := 100;
		1:
			MTBasicsPWM_0.DutyCycle := 50;
		2:
			MTBasicsPWM_0.DutyCycle := 50;
		3:
			MTBasicsPWM_0.DutyCycle := 0;
	END_CASE

	MTBasicsPWM_0(Enable := 1, Period := 1);

	doLedOn := MTBasicsPWM_0.Out AND safetyAlive;

	doLedOff := NOT doLedOn;

	diActivateAllSafetyCircuits;

	//signalization column
	doSignColumnRed := doLedOff;

	sumAuto := BOOL_TO_INT(modeZoneMagazine = modeZoneAuto) + BOOL_TO_INT(modeZonePalletization = modeZoneAuto) + BOOL_TO_INT(modeZoneOutfeed = modeZoneAuto);

	CASE sumAuto OF
		0:
			MTBasicsPWM_1.DutyCycle := 0;
		1:
			MTBasicsPWM_1.DutyCycle := 50;
		2:
			MTBasicsPWM_1.DutyCycle := 50;
		3:
			MTBasicsPWM_1.DutyCycle := 100;
	END_CASE

	MTBasicsPWM_1(Enable := 1, Period := 1);

	doSignColumnGreen := MTBasicsPWM_1.Out;

	//horn
	MTBasicsPWM_2(Enable := alarmPresent OR magazineEmpty OR interlayerSheetMagazineEmpty, DutyCycle := 50, Period := 1);

	doSignColumnOrange := MTBasicsPWM_2.Out OR bypassHorn;

	doSignColumnHorn := MTBasicsPWM_2.Out AND NOT bypassHorn;

	IF testAtAtrima THEN
		doSignColumnHorn := FALSE;
	END_IF

	IF NOT alarmPresent THEN
		bypassHorn := FALSE;
	END_IF

	IF alarmPresent AND diReset THEN
		bypassHorn := TRUE;
	END_IF

END_PROGRAM
```

### pallet_conveyors.var
```iecst
VAR
	modeConveyors : ModeConveyors;
	palletOnConveyorP13 : BOOL; (*VISU:pallet lies on conveyor*)
	palletOnConveyorP14 : BOOL;
	palletOnConveyorP15 : BOOL;
END_VAR
```

### Program Logical/plc/pallet_conveyors/pallet_conveyors (IEC) - pallet conveyors control

#### Main.st - Cyclic code
```iecst
PROGRAM _INIT
	(* Insert code here *)

END_PROGRAM

PROGRAM _CYCLIC

	readyToStart := NOT diPalletizationEDM;

	IF NOT readyToStart THEN
		modeConveyors := modeConveyorsNotReadyToStart;
	END_IF

	CASE modeConveyors OF

		modeConveyorsNotReadyToStart: //the automat is not ready to start

			IF readyToStart THEN
				modeConveyors := modeConveyorsManual;
			END_IF

		modeConveyorsManual:

			IF NOT alarmInZoneConveyors AND cmdAuto THEN
				cmdAuto := FALSE;
				modeConveyors := modeConveyorsAuto;
			END_IF
			cmdManual := FALSE;

		modeConveyorsAuto:

			IF alarmInZoneConveyors OR cmdManual THEN
				modeConveyors := modeConveyorsManual;
			END_IF

			IF palletOnConveyorP12 AND NOT palletOnConveyorP13 THEN
				cmdMovePalletP12P13 := TRUE;
			END_IF

			IF palletOnConveyorP13 AND NOT palletOnConveyorP14 THEN
				cmdMovePalletP13P14 := TRUE;
			END_IF

			IF palletOnConveyorP14 AND NOT palletOnConveyorP15 THEN
				cmdMovePalletP14P15 := TRUE;
			END_IF

	END_CASE

	//conveyor P12 + P13
	ConveyorP12P13Control;
	ConveyorP13P14Control;
	ConveyorP14P15Control;

	alarmImage[5] := NOT lightCurtainP15;
	alarmImage[8] := NOT lightCurtainP17;

	//detect if there is any alarm
	alarmInZoneConveyors := FALSE;
	FOR i:=0 TO 39 DO
		IF alarmImage[i] OR acknowledgeImage[i] THEN
			alarmInZoneConveyors := TRUE;
		END_IF
	END_FOR

END_PROGRAM
```

#### Types.typ - Local data types
```iecst
TYPE
	StateAuto :
		(
		stateAutoUndefined,
		stateAutoWaitForPallet,
		stateAutoMovePallet,
		stateAutoWaitForSensor
		);
	StateConveyor :
		(
		stateConveyorStop,
		stateConveyorWait,
		stateConveyorMoving
		);
END_TYPE
```

#### Variables.var - Local variables
```iecst
VAR
	acknowledgeImage : ARRAY[0..39] OF BOOL;
	acpI_P14 : AcpInoSdc;
	acpI_P15 : AcpInoSdc;
	alarmImage : ARRAY[0..39] OF BOOL;
	alarmInZoneConveyors : BOOL;
	cmdAuto : BOOL; (*VISU:switches pallet magazine to automatic mode*)
	cmdManual : BOOL;
	cmdMovePalletP12P13 : BOOL;
	cmdMovePalletP13P14 : BOOL;
	cmdMovePalletP14P15 : BOOL;
	diPalletSlowDownP14 : BOOL;
	diPalletStopP13 : BOOL;
	diPalletStopP14 : BOOL;
	diPalletStopP15 : BOOL;
	doConveyorP12 : BOOL; (*starts conveyor P12*)
	doConveyorP13 : BOOL;
	i : INT;
	lightCurtainP15 : BOOL;
	readyToStart : BOOL;
	stateConveyorP12P13 : StateConveyor;
	stateConveyorP13P14 : StateConveyor;
	stateConveyorP14P15 : StateConveyor;
	TON_ConveyorP12P13 : TON;
	TON_ConveyorP13P14 : TON;
	TON_ConveyorP14P15 : TON;
END_VAR
```

#### conveyorP12P13Control.st
```iecst
ACTION ConveyorP12P13Control:

	IF modeMagazine = modeMagazineNotReadyToStart THEN
		stateConveyorP12P13 := stateConveyorStop;
	END_IF

	CASE stateConveyorP12P13 OF

		stateConveyorStop:

			cmdMovePalletP12P13 := FALSE;
			doConveyorP12 := FALSE;
			doConveyorP13 := FALSE;
			stateConveyorP12P13 := stateConveyorWait;

		stateConveyorWait:

			IF cmdMovePalletP12P13 THEN
				IF palletOnConveyorP13 THEN
					alarmImage[1] := TRUE;
					stateConveyorP12P13 := stateConveyorStop;
				ELSE
					TON_ConveyorP12P13(IN := FALSE);
					stateConveyorP12P13 := stateConveyorMoving;
				END_IF
			END_IF

		stateConveyorMoving:

			doConveyorP12 := TRUE;
			doConveyorP13 := TRUE;

			//start timer
			TON_ConveyorP12P13(IN := TRUE, PT := T#12s);

			IF NOT cmdMovePalletP12P13 THEN
				stateConveyorP12P13 := stateConveyorStop;
			END_IF

			//sensor reached?
			IF palletOnConveyorP13 THEN
				palletOnConveyorP12 := FALSE;
				stateConveyorP12P13 := stateConveyorStop;
			END_IF

			//timeout?
			IF TON_ConveyorP12P13.Q THEN
				alarmImage[0] := TRUE;
				stateConveyorP12P13 := stateConveyorStop;
			END_IF

	END_CASE

	//detect pallet on conveyor
	IF diPalletStopP13 THEN
		palletOnConveyorP13 := TRUE;
	END_IF

	//edge alarms
	IF acknowledgeImage[0] THEN
		alarmImage[0] := FALSE;
	END_IF
	IF acknowledgeImage[1] THEN
		alarmImage[1] := FALSE;
	END_IF
END_ACTION
```

#### conveyorP13P14Control.st
```iecst
ACTION ConveyorP13P14Control:

	IF modeConveyors = modeConveyorsNotReadyToStart THEN
		stateConveyorP13P14 := stateConveyorStop;
	END_IF

	CASE stateConveyorP13P14 OF

		stateConveyorStop:

			cmdMovePalletP13P14 := FALSE;
			doConveyorP13 := FALSE;
			acpI_P14.switchOn := TRUE;
			acpI_P14.speed := 0;
			acpI_P14.reset := TRUE;
			stateConveyorP13P14 := stateConveyorWait;

		stateConveyorWait:

			IF cmdMovePalletP13P14 THEN
				IF palletOnConveyorP14 THEN
					alarmImage[3] := TRUE;
					stateConveyorP12P13 := stateConveyorStop;
				ELSE
					TON_ConveyorP13P14(IN := FALSE);
					stateConveyorP13P14 := stateConveyorMoving;
				END_IF
			END_IF

		stateConveyorMoving:

			doConveyorP13 := TRUE;
			acpI_P14.speed := 500;

			IF NOT cmdMovePalletP13P14 THEN
				stateConveyorP13P14 := stateConveyorStop;
			END_IF

			//sensor reached?
			IF diPalletSlowDownP14 THEN
				palletOnConveyorP13 := FALSE;
				TON_ConveyorP13P14(IN := FALSE);
				stateConveyorP13P14 := stateConveyorMovingSlow;
			END_IF

			//timeout?
			TON_ConveyorP13P14(IN := TRUE, PT := T#12s);
			IF TON_ConveyorP13P14.Q THEN
				alarmImage[4] := TRUE;
				stateConveyorP13P14 := stateConveyorStop;
			END_IF

		stateConveyorMovingSlow:

			acpI_P14.speed := 200;

			IF NOT cmdMovePalletP13P14 THEN
				stateConveyorP13P14 := stateConveyorStop;
			END_IF

			IF diPalletStopP14 THEN
				stateConveyorP13P14 := stateConveyorStop;
			END_IF

			//timeout?
			TON_ConveyorP13P14(IN := TRUE, PT := T#6s);
			IF TON_ConveyorP13P14.Q THEN
				alarmImage[2] := TRUE;
				stateConveyorP13P14 := stateConveyorStop;
			END_IF
	END_CASE

	//control of ACOPOSinverter P14
	acpI_P14();

	//detect pallet
	IF diPalletStopP14 THEN
		palletOnConveyorP14 := TRUE;
	END_IF

	//edge alarms
	IF acknowledgeImage[2] THEN
		alarmImage[2] := FALSE;
	END_IF
	IF acknowledgeImage[3] THEN
		alarmImage[3] := FALSE;
	END_IF
	IF acknowledgeImage[4] THEN
		alarmImage[4] := FALSE;
	END_IF

END_ACTION
```

#### conveyorP13Control.st - not listed in the package file held
```iecst
ACTION ConveyorP13Control:

	//detect pallet on conveyor
	IF diPalletOnConveyorP13 THEN
		palletOnConveyorP13 := TRUE;
	END_IF

END_ACTION
```

#### conveyorP14P15Control.st - not listed in the package file held
```iecst
ACTION ConveyorP14P15Control:

	IF modeConveyors = modeConveyorsNotReadyToStart THEN
		stateConveyorP14P15 := stateConveyorStop;
	END_IF

	CASE stateConveyorP14P15 OF

		stateConveyorStop:

			cmdMovePalletP14P15 := FALSE;
			acpI_P14.switchOn := TRUE;
			acpI_P14.speed := 0;
			acpI_P14.reset := TRUE;
			acpI_P15.switchOn := TRUE;
			acpI_P15.speed := 0;
			acpI_P15.reset := TRUE;
			stateConveyorP14P15 := stateConveyorWait;

		stateConveyorWait:

			IF cmdMovePalletP14P15 THEN
				IF palletOnConveyorP15 THEN
					alarmImage[6] := TRUE;
					stateConveyorP14P15 := stateConveyorStop;
				ELSE
					TON_ConveyorP14P15(IN := FALSE);
					stateConveyorP14P15 := stateConveyorMoving;
				END_IF
			END_IF

		stateConveyorMoving:

			acpI_P14.speed := 500;
			acpI_P15.speed := 500;

			IF NOT cmdMovePalletP14P15 THEN
				stateConveyorP14P15 := stateConveyorStop;
			END_IF

			//sensor reached?
			IF diPalletStopP15 THEN
				palletOnConveyorP14 := FALSE;
				stateConveyorP14P15 := stateConveyorStop;
			END_IF

			//timeout?
			TON_ConveyorP14P15(IN := TRUE, PT := T#12s);
			IF TON_ConveyorP14P15.Q THEN
				alarmImage[7] := TRUE;
				stateConveyorP14P15 := stateConveyorStop;
			END_IF

	END_CASE

	//control of ACOPOSinverter P15
	acpI_P15();

	//detect pallet
	IF diPalletStopP15 THEN
		palletOnConveyorP15 := TRUE;
	END_IF

	//edge alarms
	IF acknowledgeImage[6] THEN
		alarmImage[6] := FALSE;
	END_IF
	IF acknowledgeImage[7] THEN
		alarmImage[7] := FALSE;
	END_IF

END_ACTION
```

### pallet_outfeed.var
```iecst
VAR
	statusMessageOutfeed : INT;
END_VAR
```

### Program Logical/plc/pallet_outfeed/pallet_outfeed/pallet_outfeed

#### Main.st
```iecst
PROGRAM _INIT
	(* Insert code here *)

END_PROGRAM

PROGRAM _CYCLIC
	statusMessageOutfeed;

END_PROGRAM
```

### Program Logical/plc/pallet_outfeed/wrapper/wrapper (IEC) - wrapper control

#### Variables.var
```iecst
VAR
	diDoor2opened : BOOL;
	diOpenDoors2 : BOOL; (*button to open doors*)
	diCloseDoors2 : BOOL; (*button to close doors*)
END_VAR
```

### Program Logical/plc/pallett_magazine/pallet_magazine

#### Variables.var
```iecst
VAR
	armsState : ArmsState; (*VISU:arms state*)
	closeArms : BOOL; (*valve to close the arms*)
	cmdAutomatMode : BOOL; (*3 funkce v 1 (reset safety+ovladaci obvody + start automatu)*)
	cmdCloseArms : BOOL; (*VISU:command to close the arms*)
	cmdManualMode : BOOL; (*VISU:switches pallet magazine to manual mode*)
	cmdDown : BOOL; (*VISU:go with magazine up*)
	cmdUp : BOOL; (*VISU:go with magazine down*)
	moveToLowerPosition : BOOL; (*go with magazine to lower position*)
	moveToMiddlePosition : BOOL; (*go with magazine to middle position*)
	moveToUpperPosition : BOOL; (*go with magazine to upper position*)
	cmdOpenArms : BOOL; (*VISU:commad to open the arms*)
	leftArmClosed : BOOL; (*left arm is closed*)
	leftArmOpened : BOOL; (*left arm is opened*)
	magazineBrake : BOOL; (*1=brake released*)
	magazineDown : BOOL; (*contactor to go down*)
	magazineLooseChain : BOOL; (*lower HW end switch*)
	magazineLowerPosition : BOOL; (*magazine in lower position*)
	magazineMiddlePositon : BOOL; (*magazine in middle position*)
	magazineSafetyViolation : BOOL; (*safety violation*)
	magazineState : MagazineState;
	magazineUp : BOOL; (*contactor to go up*)
	magazineUpperHwEnd : BOOL; (*upper HW end switch*)
	magazineUpperPosition : BOOL; (*magazine in upper position*)
	modeOfOperation : ModeOfOperation;
	motorProtectionP11 : BOOL;
	openArms : BOOL; (*valve to open the arms*)
	palletOnConveyorP12 : BOOL; (*pallet detected on conveyor P12*)
	rightArmClosed : BOOL; (*right arm is closed*)
	rightArmOpened : BOOL; (*right arm is opened*)
	TON_CloseLeftRequest : TON;
	TON_CloseRightRequest : TON;
	TON_MoveToTheUpperPositon : TON;
	TON_OpenLeftRequest : TON;
	TON_OpenRightRequest : TON;
END_VAR
```

#### Main.st
```iecst
(*Control OF pallet magazine, also called "zásobník palet" nebo "stohovač" *)

PROGRAM _INIT

END_PROGRAM

PROGRAM _CYCLIC

	CASE modeOfOperation OF

		notReadyToStart: //the automat is not ready to start
			IF NOT magazineSafetyViolation AND airPresureOK THEN
				modeOfOperation := readyToStart;
			END_IF

		readyToStart:

			IF cmdManualMode OR cmdAllToManualMode THEN
				modeOfOperation := manualMode;
			END_IF

		manualMode:

			MagazineControl;

	END_CASE;

	//action to control the arms
	ArmsControl;

	(* error detection *)
	IF magazineSafetyViolation THEN
		MpAlarmXSet(gAlarmXCore,'PalletMagazineSafetyViolation');
	ELSE
		MpAlarmXReset(gAlarmXCore,'PalletMagazineSafetyViolation');
	END_IF

	IF NOT motorProtectionP11 THEN
		MpAlarmXSet(gAlarmXCore,'MotorProtectionP11');
	ELSE
		MpAlarmXReset(gAlarmXCore,'MotorProtectionP11');
	END_IF

END_PROGRAM
```

### Program Logical/plc/product_infeed/product_infeed (IEC) - product infeed control

#### Main.st - Cyclic code
```iecst
PROGRAM _INIT
	(* Insert code here *)

END_PROGRAM

PROGRAM _CYCLIC
	diDoor1opened;
	diOpenDoors1;
	diCloseDoors1;

END_PROGRAM
```

### Program Logical/plc/robot_control/robot_control (IEC) - robot control

#### Main.st
```iecst
PROGRAM _INIT
	(* Insert code here *)

END_PROGRAM

PROGRAM _CYCLIC

END_PROGRAM
```

### Program Logical/plc/wrapper/wrapper (IEC) - wrapper control

#### Main.st
```iecst
PROGRAM _INIT
	(* Insert code here *)

END_PROGRAM

PROGRAM _CYCLIC
	diDoor2opened;
	diOpenDoors2;
	diCloseDoors2;

END_PROGRAM
```

- Visualisation Logical/visualization (not shown)

### Package Logical/AsSafetySolution - AsSafety design sample

### Program Logical/AsSafetySolution/SafetySample (IEC) - Handling

#### SafetySample.st - Implementation code
```iecst
(********************************************************************
 * COPYRIGHT -- Bernecker + Rainer
 ********************************************************************
 * Program: SafetySample
 * File: SafetySample.st
 * Author: B&R
 ********************************************************************
 * Implementation of program SafetySample
 ********************************************************************)

PROGRAM _INIT

(* command structure for remote control FUB *)
remotecmd.Version := safeVERSION_R107;	(* version *)
remotecmd.Password := '123456';				(* password *)

(* command structure for application download *)
appcmd1.Version := safeVERSION_R107;	(* version *)
appcmd1.Password := '123456';					(* password *)
appcmd1.ApplicationID := 1;				(* application id *)

(* command structure for machine options download *)
datacmd1.Version := safeVERSION_R107;								(* version *)
datacmd1.Password := '123456';											(* password *)
datacmd1.pDeviceListInput := ADR(visuDeviceListInput);				(* device list *)
datacmd1.pMachineOptionsInput := ADR(dataMachineOptionsBitInput);	(* bit machine options *)
datacmd1.pModuleFlagsInput := ADR(dataModuleFlagsInput);			(* module flags *)
datacmd1.pAcknMachineOptions := ADR(dataAcknMachineOptions);		(* acknowledge information *)

(* command structure for extended machine options *)
datacmd2.Version := safeVERSION_R107;					(* version *)
datacmd2.Password := '123456';								(* password *)
datacmd2.pIntDataInput := ADR(visuIntInput);			(* INT channels *)
datacmd2.NumberIntInput := 1;							(* number of INT channels *)
datacmd2.pUintDataInput := ADR(visuUintInput);			(* UINT channels *)
datacmd2.NumberUintInput := 1;							(* number of UINT channels *)
datacmd2.pDintDataInput := ADR(visuDintInput);			(* DINT channels *)
datacmd2.NumberDintInput := 1;							(* number of DINT channels *)
datacmd2.pUdintDataInput := ADR(visuUdintInput);		(* UDINT channels *)
datacmd2.NumberUdintInput := 1;							(* number of UDINT channels *)
datacmd2.pAcknMachineOptions := ADR(visuAcknExtData);	(* acknowledge information *)

(* hide elements in visualization *)
FOR xcnt := 0 TO SIZEOF(statusButtonActiv) - 1 DO
	statusButtonActiv[xcnt] := 1;
END_FOR

(* hide elements in visualization *)
statusButtonUnlockApp := 1;
statusButtonUnlockData := 1;
statusAcknInfoData := 1;
statusButtonUnlockExtData := 1;
statusAcknInfoExtData := 1;
statusDialog := 1;

(* set SafeLOGIC ID *)
visuUsedSLIDRemote := 1;
visuUsedSLIDData := 1;

END_PROGRAM

PROGRAM _CYCLIC
	(****************************************************************************************************************************************)
	(****************************************************************************************************************************************)
	(****************************************************************************************************************************************)
	(* show dialog to ackn command *)
	IF (dialogRemoteCmd = 1) THEN
		statusDialog := 0;
		dialogRemoteCmd := 0;
		indexButtonLeft := 0;
		indexButtonRight := 1;
		indexHeaderText := 0;
		IF (remotecmd.Data = safeCMD_SK_FORMAT) THEN
			indexMessageText := 0;
		ELSIF (remotecmd.Data = safeCMD_SK_XCHG) THEN
			indexMessageText := 1;
		ELSIF (remotecmd.Data = safeCMD_1_UDID_ACKN) THEN
			indexMessageText := 2;
		ELSIF (remotecmd.Data = safeCMD_2_UDID_ACKN) THEN
			indexMessageText := 3;
		ELSIF (remotecmd.Data = safeCMD_3_UDID_ACKN) THEN
			indexMessageText := 4;
		ELSIF (remotecmd.Data = safeCMD_4_UDID_ACKN) THEN
			indexMessageText := 5;
		ELSIF (remotecmd.Data =  safeCMD_N_UDID_ACKN) THEN
			indexMessageText := 6;
		ELSIF (remotecmd.Data =  safeCMD_CLEAR_DATA) THEN
			indexMessageText := 7;
		ELSIF (remotecmd.Data = safeCMD_FW_ACKN) THEN
			indexMessageText := 8;
		ELSIF (remotecmd.Data = safeCMD_RESET) THEN
			indexMessageText := 9;
		END_IF
	END_IF

	(* if dialog is ackn execute fub *)
	IF (dialogButtonLeft = 1 AND indexHeaderText = 0) THEN
		executeRemoteCmd := 1;
		dialogButtonLeft := 0;
		statusDialog := 1;
	ELSIF (dialogButtonRight = 1 AND indexHeaderText = 0) THEN
		dialogButtonRight := 0;
		statusDialog := 1;
	END_IF

	(* password must be at least 6 characters long *)
	IF brsstrlen(ADR(remotecmd.NewPassword)) < 6 THEN
		statusSetPassword := 2;
	ELSE
		statusSetPassword := 0;
	END_IF

	safeRemoteControl_0(SafeLOGICID := visuUsedSLIDRemote, Execute := executeRemoteCmd, pCommandData := ADR(remotecmd));
	(* reset execution flag *)
	IF (safeRemoteControl_0.Done = 1 OR safeRemoteControl_0.Error = 1) THEN
		executeRemoteCmd := 0;
	END_IF

	(* variables for visualization *)
	IF (safeRemoteControl_0.SafeLOGICStatus.SafeKEYChanged = 1) THEN
		FOR xcnt := 0 TO SIZEOF(statusButtonActiv) - 1 DO
			statusButtonActiv[xcnt] := 1;
 			statusButtonInactiv[xcnt] := 0;
		END_FOR
		statusButtonActiv[1] := 0;
 		statusButtonInactiv[1] := 1;
	ELSIF (safeRemoteControl_0.SafeLOGICStatus.NumberOfUDIDMismatches = 1 AND safeRemoteControl_0.SafeLOGICStatus.Scanning = 0) THEN
		FOR xcnt := 0 TO SIZEOF(statusButtonActiv) - 1 DO
			statusButtonActiv[xcnt] := 1;
 			statusButtonInactiv[xcnt] := 0;
		END_FOR
		statusButtonActiv[3] := 0;
 		statusButtonInactiv[3] := 1;
	ELSIF (safeRemoteControl_0.SafeLOGICStatus.NumberOfUDIDMismatches = 2 AND safeRemoteControl_0.SafeLOGICStatus.Scanning = 0) THEN
		FOR xcnt := 0 TO SIZEOF(statusButtonActiv) - 1 DO
			statusButtonActiv[xcnt] := 1;
 			statusButtonInactiv[xcnt] := 0;
		END_FOR
		statusButtonActiv[4] := 0;
 		statusButtonInactiv[4] := 1;
	ELSIF (safeRemoteControl_0.SafeLOGICStatus.NumberOfUDIDMismatches = 3 AND safeRemoteControl_0.SafeLOGICStatus.Scanning = 0) THEN
		FOR xcnt := 0 TO SIZEOF(statusButtonActiv) - 1 DO
			statusButtonActiv[xcnt] := 1;
 			statusButtonInactiv[xcnt] := 0;
		END_FOR
		statusButtonActiv[5] := 0;
 		statusButtonInactiv[5] := 1;
	ELSIF (safeRemoteControl_0.SafeLOGICStatus.NumberOfUDIDMismatches = 4 AND safeRemoteControl_0.SafeLOGICStatus.Scanning = 0) THEN
		FOR xcnt := 0 TO SIZEOF(statusButtonActiv) - 1 DO
			statusButtonActiv[xcnt] := 1;
 			statusButtonInactiv[xcnt] := 0;
		END_FOR
		statusButtonActiv[6] := 0;
 		statusButtonInactiv[6] := 1;
	ELSIF (safeRemoteControl_0.SafeLOGICStatus.NumberOfUDIDMismatches > 4 AND safeRemoteControl_0.SafeLOGICStatus.Scanning = 0) THEN
		FOR xcnt := 0 TO SIZEOF(statusButtonActiv) - 1 DO
			statusButtonActiv[xcnt] := 1;
 			statusButtonInactiv[xcnt] := 0;
		END_FOR
		statusButtonActiv[7] := 0;
 		statusButtonInactiv[7] := 1;
	ELSIF (safeRemoteControl_0.SafeLOGICStatus.NumberOfDifferentFirmware <> 0 AND safeRemoteControl_0.SafeLOGICStatus.Scanning = 0) THEN
		FOR xcnt := 0 TO SIZEOF(statusButtonActiv) - 1 DO
			statusButtonActiv[xcnt] := 1;
 			statusButtonInactiv[xcnt] := 0;
		END_FOR
		statusButtonActiv[11] := 0;
 		statusButtonInactiv[11] := 1;
	ELSE
		FOR xcnt := 0 TO SIZEOF(statusButtonActiv) - 1 DO
			statusButtonActiv[xcnt] := 1;
 			statusButtonInactiv[xcnt] := 0;
		END_FOR
	END_IF
	(* status text - MXCHG *)
	IF (safeRemoteControl_0.SafeLOGICStatus.LedTestActive = 1) THEN
		indexMxchgLed := 40;
	ELSIF (safeRemoteControl_0.SafeLOGICStatus.Scanning = 1) THEN
		indexMxchgLed := 30;
	ELSIF (safeRemoteControl_0.SafeLOGICStatus.NumberOfUDIDMismatches = 1) THEN
		indexMxchgLed := 1;
	ELSIF (safeRemoteControl_0.SafeLOGICStatus.NumberOfUDIDMismatches = 2) THEN
		indexMxchgLed := 2;
	ELSIF (safeRemoteControl_0.SafeLOGICStatus.NumberOfUDIDMismatches = 3) THEN
		indexMxchgLed := 3;
	ELSIF (safeRemoteControl_0.SafeLOGICStatus.NumberOfUDIDMismatches = 4) THEN
		indexMxchgLed := 4;
	ELSIF (safeRemoteControl_0.SafeLOGICStatus.NumberOfUDIDMismatches > 4) THEN
		indexMxchgLed := 5;
	ELSIF (safeRemoteControl_0.SafeLOGICStatus.NumberOfMissingModules <> 0) THEN
		indexMxchgLed := 20;
	ELSIF (safeRemoteControl_0.SafeLOGICStatus.NumberOfUDIDMismatches = 0) THEN
		indexMxchgLed := 10;
	END_IF
	(* status text - FW-ACKN *)
	IF (safeRemoteControl_0.SafeLOGICStatus.SafeKEYChanged = 0 AND safeRemoteControl_0.SafeLOGICStatus.NumberOfDifferentFirmware = 0) THEN
		indexFwAcknLed := 10;
	ELSIF (safeRemoteControl_0.SafeLOGICStatus.SafeKEYChanged = 1) THEN
		indexFwAcknLed := 1;
	ELSIF (safeRemoteControl_0.SafeLOGICStatus.NumberOfDifferentFirmware <> 0) THEN
		indexFwAcknLed := 2;
	END_IF
	(* status text - FAIL *)
	IF (safeRemoteControl_0.SafeLOGICStatus.FailSafe <> 16#55) THEN
		indexFAILLed := 2;
	ELSIF (safeRemoteControl_0.SafeLOGICStatus.openSAFETYstate = 0) THEN
		indexFAILLed := 0;
	ELSIF (safeRemoteControl_0.SafeLOGICStatus.openSAFETYstate = 1) THEN
		indexFAILLed := 1;
	END_IF
	(* status text - R/E *)
	indexRELed := safeRemoteControl_0.SafeLOGICStatus.SafeOSState;

	(****************************************************************************************************************************************)
	(****************************************************************************************************************************************)
	(****************************************************************************************************************************************)
	(* show dialog to ackn command *)
	IF (dialogApplication = 1) THEN
		statusDialog := 0;
		dialogApplication := 0;
		indexButtonLeft := 0;
		indexButtonRight := 1;
		indexHeaderText := 1;
		indexMessageText := 10;
	END_IF

	(* if dialog is ackn unlock application *)
	IF (dialogButtonLeft = 1 AND indexHeaderText = 1) THEN
		appcmd1.Unlock := 1;
		dialogButtonLeft := 0;
		statusDialog := 1;
	ELSIF (dialogButtonRight = 1 AND indexHeaderText = 1) THEN
		appcmd1.Unlock := 2;
		dialogButtonRight := 0;
		statusDialog := 1;
	END_IF

	(* convert application CRC to HEX string *)
	itoahex(safeDownloadApplication_0.ApplicationCRC, ADR(visuApplicationCRC));

	safeDownloadApplication_0(SafeLOGICID := appcmd1.ApplicationID, Execute := executeapp1, pCommandData := ADR(appcmd1));

	(* show unlock button *)
	IF (safeDownloadApplication_0.UnlockRequired = 1) THEN
		statusButtonUnlockApp := 0;
	ELSE
		appcmd1.Unlock := 0;
		statusButtonUnlockApp := 1;
	END_IF

	(****************************************************************************************************************************************)
	(****************************************************************************************************************************************)
	(****************************************************************************************************************************************)
	(* disable machine options *)
	IF (visuEnableMachineOptions = FALSE) THEN
		datacmd1.pMachineOptionsInput := 0;
	ELSE
		datacmd1.pMachineOptionsInput := ADR(dataMachineOptionsBitInput);
	END_IF

	(* disable module flags *)
	IF (visuEnableModuleFlags = FALSE) THEN
		datacmd1.pModuleFlagsInput := 0;
	ELSE
		datacmd1.pModuleFlagsInput := ADR(dataModuleFlagsInput);
	END_IF

	(* Machine Option Bit #000 *)
	IF (visuMachineOptionsBitInput[0] = 1) THEN
		dataMachineOptionsBitInput.BitData[0].0 := 1;
	ELSE
		dataMachineOptionsBitInput.BitData[0].0 := 0;
	END_IF
	(* Machine Option Bit #001 *)
	IF (visuMachineOptionsBitInput[1] = 1) THEN
		dataMachineOptionsBitInput.BitData[0].1 := 1;
	ELSE
		dataMachineOptionsBitInput.BitData[0].1 := 0;
	END_IF
	(* Machine Option Bit #002 *)
	IF (visuMachineOptionsBitInput[2] = 1) THEN
		dataMachineOptionsBitInput.BitData[0].2 := 1;
	ELSE
		dataMachineOptionsBitInput.BitData[0].2 := 0;
	END_IF
	(* Optional Flag Module #1 *)
	IF (visuModuleFlagsOptionalInput[1] = 1) THEN
		dataModuleFlagsInput.Optional[0].1 := 1;
	ELSE
		dataModuleFlagsInput.Optional[0].1 := 0;
	END_IF
	(* Optional Flag Module #2 *)
	IF (visuModuleFlagsOptionalInput[2] = 1) THEN
		dataModuleFlagsInput.Optional[0].2 := 1;
	ELSE
		dataModuleFlagsInput.Optional[0].2 := 0;
	END_IF
	(* Startup Flag Module #1 *)
	IF (visuModuleFlagsStartupInput[1] = 1) THEN
		dataModuleFlagsInput.Startup[0].1 := 1;
	ELSE
		dataModuleFlagsInput.Startup[0].1 := 0;
	END_IF
	(* Startup Flag Module #2 *)
	IF (visuModuleFlagsStartupInput[2] = 1) THEN
		dataModuleFlagsInput.Startup[0].2 := 1;
	ELSE
		dataModuleFlagsInput.Startup[0].2 := 0;
	END_IF
	(* Not_Present Flag Module #1 *)
	IF (visuModuleFlagsNotPresentInput[1] = 1) THEN
		dataModuleFlagsInput.NotPresent[0].1 := 1;
	ELSE
		dataModuleFlagsInput.NotPresent[0].1 := 0;
	END_IF
	(* Not_Present Flag Module #2 *)
	IF (visuModuleFlagsNotPresentInput[2] = 1) THEN
		dataModuleFlagsInput.NotPresent[0].2 := 1;
	ELSE
		dataModuleFlagsInput.NotPresent[0].2 := 0;
	END_IF

	(* Ackn Machine Option Bit #000 *)
	IF (visuAcknMachineOptions[0] = 1) THEN
		dataAcknMachineOptions.AcknBitOptions[0].0 := 1;
	ELSE
		dataAcknMachineOptions.AcknBitOptions[0].0 := 0;
	END_IF
	(* Ackn Machine Option Bit #001 *)
	IF (visuAcknMachineOptions[1] = 1) THEN
		dataAcknMachineOptions.AcknBitOptions[0].1 := 1;
	ELSE
		dataAcknMachineOptions.AcknBitOptions[0].1 := 0;
	END_IF
	(* Ackn Machine Option Bit #002 *)
	IF (visuAcknMachineOptions[2] = 1) THEN
		dataAcknMachineOptions.AcknBitOptions[0].2 := 1;
	ELSE
		dataAcknMachineOptions.AcknBitOptions[0].2 := 0;
	END_IF

	(* show dialog to ackn command *)
	IF (dialogData = 1) THEN
		statusDialog := 0;
		dialogData := 0;
		indexButtonLeft := 0;
		indexButtonRight := 1;
		indexHeaderText := 2;
		indexMessageText := 11;
	END_IF

	(* if dialog is ackn unlock data *)
	IF (dialogButtonLeft = 1 AND indexHeaderText = 2) THEN
		datacmd1.Unlock := 1;
		dialogButtonLeft := 0;
		statusDialog := 1;
	ELSIF (dialogButtonRight = 1 AND indexHeaderText = 2) THEN
		datacmd1.Unlock := 2;
		dialogButtonRight := 0;
		statusDialog := 1;
	END_IF

	safeDownloadData_0(SafeLOGICID := visuUsedSLIDData, Execute := executedata1, Type:= safeDATA_TYPE_MAOP, pCommandData := ADR(datacmd1));

	(* data compare failed *)
	IF (safeDownloadData_0.StatusID = safeERR_DL_COMPARE_FAILED) THEN
		indexCompareTextData := 2;
	ELSE
		indexCompareTextData := 0;
	END_IF

	IF (safeDownloadData_0.UnlockRequired = 1) THEN
		(* data compare successful *)
		indexCompareTextData := 1;
		IF (datacmd1.pDeviceListOutput <> 0 AND datacmd1.NumberDevicesOutput <> 0) THEN
			pDeviceListOut ACCESS datacmd1.pDeviceListOutput;

			(* device #1 *)
			visuDeviceListOutput[0].SADR := pDeviceListOut[0].SADR;
			brsmemcpy(ADR(visuDeviceListOutput[0].UDID_High), ADR(pDeviceListOut[0].UDID[0]), 2);
			(* swap UDID *)
			visuDeviceListOutput[0].UDID_High := swapUINT(visuDeviceListOutput[0].UDID_High);
			brsmemcpy(ADR(visuDeviceListOutput[0].UDID_Low), ADR(pDeviceListOut[0].UDID[2]), 4);
			(* swap UDID *)
			visuDeviceListOutput[0].UDID_Low := swapUDINT(visuDeviceListOutput[0].UDID_Low);
			(* device #2 *)
			visuDeviceListOutput[1].SADR := pDeviceListOut[1].SADR;
			brsmemcpy(ADR(visuDeviceListOutput[1].UDID_High), ADR(pDeviceListOut[1].UDID[0]), 2);
			(* swap UDID *)
			visuDeviceListOutput[1].UDID_High := swapUINT(visuDeviceListOutput[1].UDID_High);
			brsmemcpy(ADR(visuDeviceListOutput[1].UDID_Low), ADR(pDeviceListOut[1].UDID[2]), 4);
			(* swap UDID *)
			visuDeviceListOutput[1].UDID_Low := swapUDINT(visuDeviceListOutput[1].UDID_Low);
		END_IF

		IF (datacmd1.pMachineOptionsOutput <> 0) THEN
			pMachineOptionsBitOut ACCESS datacmd1.pMachineOptionsOutput;

			(* Machine Option Bit #000 *)
			IF (pMachineOptionsBitOut.BitData[0].0 = 1) THEN
				visuMachineOptionsBitOutput[0] := 1;
			END_IF
			(* Machine Option Bit #001 *)
			IF (pMachineOptionsBitOut.BitData[0].1 = 1) THEN
				visuMachineOptionsBitOutput[1] := 1;
			END_IF
			(* Machine Option Bit #002 *)
			IF (pMachineOptionsBitOut.BitData[0].2 = 1) THEN
				visuMachineOptionsBitOutput[2] := 1;
			END_IF
		END_IF

		IF (datacmd1.pModuleFlagsOutput <> 0) THEN
			pModuleFlagsOut ACCESS datacmd1.pModuleFlagsOutput;

			(* Optional Flag Module #1 *)
			IF (pModuleFlagsOut.Optional[0].1 = 1) THEN
				visuModuleFlagsOptionalOutput[1] := 1;
			END_IF
			(* Optional Flag Module #2 *)
			IF (pModuleFlagsOut.Optional[0].2 = 1) THEN
				visuModuleFlagsOptionalOutput[2] := 1;
			END_IF
			(* Startup Flag Module #1 *)
			IF (pModuleFlagsOut.Startup[0].1 = 1) THEN
				visuModuleFlagsStartupOutput[1] := 1;
			END_IF
			(* Startup Flag Module #2 *)
			IF (pModuleFlagsOut.Startup[0].2 = 1) THEN
				visuModuleFlagsStartupOutput[2] := 1;
			END_IF
			(* Not_Present Flag Module #1 *)
			IF (pModuleFlagsOut.NotPresent[0].1 = 1) THEN
				visuModuleFlagsNotPresentOutput[1] := 1;
			END_IF
			(* Not_Present Flag Module #2 *)
			IF (pModuleFlagsOut.NotPresent[0].2 = 1) THEN
				visuModuleFlagsNotPresentOutput[2] := 1;
			END_IF
		END_IF
		(* show ackn box *)
		statusAcknInfoData := 0;
		(* show unlock button unlocked if one ACK is set *)
		IF (visuAcknMachineOptions[0] = 1 OR visuAcknMachineOptions[1] = 1 OR visuAcknMachineOptions[2] = 1) THEN
			statusButtonUnlockData := 0;
		END_IF
	ELSIF (safeDownloadData_0.Done = 1 OR safeDownloadData_0.Error = 1) THEN
		(* reset visualization elements *)
		brsmemset(ADR(visuDeviceListOutput), 0, SIZEOF(visuDeviceListOutput));
		brsmemset(ADR(visuMachineOptionsBitOutput), 0, SIZEOF(visuMachineOptionsBitOutput));
		brsmemset(ADR(visuModuleFlagsOptionalOutput), 0, SIZEOF(visuModuleFlagsOptionalOutput));
		brsmemset(ADR(visuModuleFlagsStartupOutput), 0, SIZEOF(visuModuleFlagsStartupOutput));
		brsmemset(ADR(visuModuleFlagsNotPresentOutput), 0, SIZEOF(visuModuleFlagsNotPresentOutput));
		(* hide ackn box *)
		statusAcknInfoData := 1;
		(* hide unlock button *)
		datacmd1.Unlock := 0;
		statusButtonUnlockData := 1;
		(* reset ackn flags *)
		visuAcknMachineOptions[0] := 0;
		visuAcknMachineOptions[1] := 0;
		visuAcknMachineOptions[2] := 0;
	ELSE
		(* hide ackn box *)
		statusAcknInfoData := 1;
		(* hide unlock button *)
		datacmd1.Unlock := 0;
		statusButtonUnlockData := 1;
	END_IF

	(****************************************************************************************************************************************)
	(****************************************************************************************************************************************)
	(****************************************************************************************************************************************)
	(* Enable for INT set *)
	IF (visuEnableINTOptions <> 0) THEN
		datacmd2.pIntDataInput := ADR(visuIntInput);
		datacmd2.NumberIntInput := 1;
	ELSE
		datacmd2.pIntDataInput := 0;
		datacmd2.NumberIntInput := 0;
	END_IF
	(* Enable for UINT set *)
	IF (visuEnableUINTOptions <> 0) THEN
		datacmd2.pUintDataInput := ADR(visuUintInput);
		datacmd2.NumberUintInput := 1;
	ELSE
		datacmd2.pUintDataInput := 0;
		datacmd2.NumberUintInput := 0;
	END_IF
	(* Enable for DINT set *)
	IF (visuEnableDINTOptions <> 0) THEN
		datacmd2.pDintDataInput := ADR(visuDintInput);
		datacmd2.NumberDintInput := 1;
	ELSE
		datacmd2.pDintDataInput := 0;
		datacmd2.NumberDintInput := 0;
	END_IF
	(* Enable for UDINT set *)
	IF (visuEnableUDINTOptions <> 0) THEN
		datacmd2.pUdintDataInput := ADR(visuUdintInput);
		datacmd2.NumberUdintInput := 1;
	ELSE
		datacmd2.pUdintDataInput := 0;
		datacmd2.NumberUdintInput := 0;
	END_IF

	(* show dialog to ackn command *)
	IF (dialogExtData = 1) THEN
		statusDialog := 0;
		dialogExtData := 0;
		indexButtonLeft := 0;
		indexButtonRight := 1;
		indexHeaderText := 3;
		indexMessageText := 11;
	END_IF

	(* if dialog is ackn unlock data *)
	IF (dialogButtonLeft = 1 AND indexHeaderText = 3) THEN
		datacmd2.Unlock := 1;
		dialogButtonLeft := 0;
		statusDialog := 1;
	ELSIF (dialogButtonRight = 1 AND indexHeaderText = 3) THEN
		datacmd2.Unlock := 2;
		dialogButtonRight := 0;
		statusDialog := 1;
	END_IF

	safeDownloadData_1(SafeLOGICID := visuUsedSLIDData, Execute := executedata2, Type:= safeDATA_TYPE_EXTMAOP, pCommandData := ADR(datacmd2));

	(* data compare failed *)
	IF (safeDownloadData_1.StatusID = safeERR_DL_COMPARE_FAILED) THEN
		indexCompareTextExtData := 2;
	ELSE
		indexCompareTextExtData := 0;
	END_IF

	IF (safeDownloadData_1.UnlockRequired = 1) THEN
		(* data compare successful *)
		indexCompareTextExtData := 1;

		(* INT channels *)
		IF (datacmd2.pIntDataOutput <> 0 AND datacmd2.NumberIntOutput <> 0) THEN
			brsmemcpy(ADR(visuIntOutput), datacmd2.pIntDataOutput, SIZEOF(visuIntOutput));
		END_IF
		(* UINT channels *)
		IF (datacmd2.pUintDataOutput <> 0 AND datacmd2.NumberUintOutput <> 0) THEN
			brsmemcpy(ADR(visuUintOutput), datacmd2.pUintDataOutput, SIZEOF(visuUintOutput));
		END_IF
		(* DINT channels *)
		IF (datacmd2.pDintDataOutput <> 0 AND datacmd2.NumberDintOutput <> 0) THEN
			brsmemcpy(ADR(visuDintOutput), datacmd2.pDintDataOutput, SIZEOF(visuDintOutput));
		END_IF
		(* UDINT channels *)
		IF (datacmd2.pUdintDataOutput <> 0 AND datacmd2.NumberUdintOutput <> 0) THEN
			brsmemcpy(ADR(visuUdintOutput), datacmd2.pUdintDataOutput, SIZEOF(visuUdintOutput));
		END_IF
		(* show ackn box *)
		statusAcknInfoExtData := 0;
		(* show unlock button if one ACK is set *)
		IF (visuAcknExtData.AcknIntOptions[0] = 1 OR visuAcknExtData.AcknUintOptions[0] = 1 OR visuAcknExtData.AcknDintOptions[0] = 1 OR visuAcknExtData.AcknUdintOptions[0] = 1) THEN
			statusButtonUnlockExtData := 0;
		END_IF
	ELSIF (safeDownloadData_1.Done = 1 OR safeDownloadData_1.Error = 1) THEN
		(* reset visualization elements *)
		brsmemset(ADR(visuIntOutput), 0, SIZEOF(visuIntOutput));
		brsmemset(ADR(visuUintOutput), 0, SIZEOF(visuUintOutput));
		brsmemset(ADR(visuDintOutput), 0, SIZEOF(visuDintOutput));
		brsmemset(ADR(visuUdintOutput), 0, SIZEOF(visuUdintOutput));
		(* hide ackn box *)
		statusAcknInfoExtData := 1;
		(* hide unlock button *)
		datacmd2.Unlock := 0;
		statusButtonUnlockExtData := 1;
		(* reset ackn flags *)
		visuAcknExtData.AcknIntOptions[0] := 0;
		visuAcknExtData.AcknUintOptions[0] := 0;
		visuAcknExtData.AcknDintOptions[0] := 0;
		visuAcknExtData.AcknUdintOptions[0] := 0;
	ELSE
		(* hide ackn box *)
		statusAcknInfoExtData := 1;
		(* hide unlock button *)
		datacmd2.Unlock := 0;
		statusButtonUnlockExtData := 1;
	END_IF

	(****************************************************************************************************************************************)
	(****************************************************************************************************************************************)
	(****************************************************************************************************************************************)
	(* read UDID from SafeLOGIC-X *)
	IF slxused = 1 THEN
		readUDIDlowSLX(enable := 1, pDeviceName := ADR(Station), pChannelName := ADR('UDID_low'));

		IF readUDIDlowSLX.status = 0 THEN
			UDID_Low := readUDIDlowSLX.value;
		ELSIF readUDIDlowSLX.status <> 65535 THEN
			UDID_Low := 0;
		END_IF

		readUDIDhighSLX(enable := 1, pDeviceName := ADR(Station), pChannelName := ADR('UDID_high'));

		IF readUDIDhighSLX.status = 0 THEN
			UDID_High := UDINT_TO_UINT(readUDIDhighSLX.value);
		ELSIF readUDIDhighSLX.status <> 65535 THEN
			UDID_High := 0;
		END_IF

		(* hide / show visualization elements *)
		stautsSLXInformation := 0;
		statusSLInformation := 1;
	(* read UDID form SafeLOGIC *)
	ELSE
		readUDIDlowSL(enable := 1, pDevice := ADR(Interface), node := Node, index := 16#2000, subindex := 6, pData := ADR(UDID_Low), datalen := SIZEOF(UDID_Low));

		IF readUDIDlowSL.status <> 0 AND readUDIDlowSL.status <> 65535 THEN
			UDID_Low := 0;
		END_IF

		readUDIDhighSL(enable := 1, pDevice := ADR(Interface), node := Node, index := 16#2000, subindex := 7, pData := ADR(UDID_High), datalen := SIZEOF(UDID_High));

		IF readUDIDhighSL.status <> 0 AND readUDIDhighSL.status <> 65535 THEN
			UDID_High := 0;
		END_IF

		(* hide / show visualization elements *)
		stautsSLXInformation := 1;
		statusSLInformation := 0;
	END_IF

	(* convert UDID to HEX string *)
	itoahex(UDID_Low, ADR(visuUDID_Low));
	itoahex(UDID_High, ADR(visuUDID_High));

	(****************************************************************************************************************************************)
	(****************************************************************************************************************************************)
	(****************************************************************************************************************************************)
	(* write UDID for SafeLOGIC to command structure *)
	appcmd1.UDID_Low := UDID_Low;
	appcmd1.UDID_High := UDID_High;
	datacmd1.UDID_Low := UDID_Low;
	datacmd1.UDID_High := UDID_High;
	datacmd2.UDID_Low := UDID_Low;
	datacmd2.UDID_High := UDID_High;

END_PROGRAM
```

#### SafetySample.var - Local variables
```iecst
(********************************************************************
 * COPYRIGHT -- Bernecker + Rainer
 ********************************************************************
 * Program: SafetySample
 * File: SafetySample.var
 * Author: B&R
 ********************************************************************
 * Local variables of program SafetySample
 ********************************************************************)
VAR
	appcmd1 : DownloadCmdApplicationTypeV1; (*command structure for application download*)
	dataAcknMachineOptions : DownloadAcknMaOpTypeV1; (*data to acknowledge bit machine options*)
	datacmd1 : DownloadCmdMaOpTypeV1; (*command structure for machine options download*)
	datacmd2 : DownloadCmdExtMaOpTypeV1; (*command structure for extended machine options download*)
	dataMachineOptionsBitInput : ConfigurationBitOptionsTypeV1; (*data for bit machine options*)
	dataModuleFlagsInput : ConfigurationModuleFlagsTypeV1; (*data for module flags*)
	dialogApplication : BOOL; (*visualization dialog for application download*)
	dialogButtonLeft : BOOL; (*left button in visualization dialog*)
	dialogButtonRight : BOOL; (*right button in visualization dialog*)
	dialogData : BOOL; (*visualization dialog for machine options download*)
	dialogExtData : BOOL; (*visualization dialog for extended machine options download*)
	dialogRemoteCmd : BOOL; (*visualization dialog for remote control*)
	executeapp1 : BOOL; (*execute application download*)
	executedata1 : BOOL; (*execute machine options download*)
	executedata2 : BOOL; (*execute extended machine options download*)
	executeRemoteCmd : BOOL; (*execute remote control*)
	indexButtonLeft : UINT; (*index for button text*)
	indexButtonRight : UINT; (* index for button text*)
	indexCompareTextData : UINT; (*index for compare message machine options*)
	indexCompareTextExtData : UINT; (*index for compare message extended machine options*)
	indexFAILLed : UINT; (*index FAIL led*)
	indexFwAcknLed : UINT; (*index FW-ACKN led*)
	indexHeaderText : UINT; (*index dialog header text*)
	indexMessageText : UINT; (*index message text*)
	indexMxchgLed : UINT; (*index MXCHG led*)
	indexRELed : UINT; (*index R/E led*)
	Interface : STRING[80] := 'IF3'; (*interface information for SafeLOGIC*)
	Node : USINT := 1; (*node information for SafeLOGIC*)
	pDeviceListOut : REFERENCE TO ARRAY[0..1] OF ConfigurationDeviceTypeV1; (*device list from FUB*)
	pMachineOptionsBitOut : REFERENCE TO ConfigurationBitOptionsTypeV1; (*bit machine options from FUB*)
	pModuleFlagsOut : REFERENCE TO ConfigurationModuleFlagsTypeV1; (*module flags form FUB*)
	readUDIDhighSL : EplSDORead; (*function block to read UDID high from device*)
	readUDIDhighSLX : AsIOAccRead; (*function block to read UDID high from device*)
	readUDIDlowSL : EplSDORead; (*function block to read UDID low from device*)
	readUDIDlowSLX : AsIOAccRead; (*function block to read UDID low from device*)
	remotecmd : RemoteControlCmdTypeV1; (*command structure for remote control*)
	safeDownloadApplication_0 : safeDownloadApplication; (*function block safeDownloadApplication*)
	safeDownloadData_0 : safeDownloadData; (*function block safeDownloadData*)
	safeDownloadData_1 : safeDownloadData; (*function block safeDownloadData*)
	safeRemoteControl_0 : safeRemoteControl; (*function block safeRemoteControl*)
	slxused : BOOL; (*SafeLOGIC-X is used*)
	Station : STRING[80] := 'IF6.ST3'; (*station information for SafeLOGIC-X*)
	statusAcknInfoData : UINT; (*acknowledge boxes for machine options*)
	statusAcknInfoExtData : UINT; (*acknowledge boxes for extended machine options*)
	statusButtonActiv : ARRAY[0..15] OF USINT; (*button activ*)
	statusButtonInactiv : ARRAY[0..15] OF USINT; (*button inactiv*)
	statusButtonUnlockApp : UINT; (*unlock buttons application*)
	statusButtonUnlockData : UINT; (*unlock buttons data*)
	statusButtonUnlockExtData : UINT; (*unlock buttons extended data*)
	statusDialog : UINT; (*dialog box*)
	statusSetPassword : UINT; (*visualization status to set password*)
	statusSLInformation : UINT; (*display information for SafeLOGIC*)
	stautsSLXInformation : UINT; (*display information for SafeLOGIC-X*)
	UDID_High : UINT; (*UDID_high for SafelOGIC*)
	UDID_Low : UDINT; (*UDID_low for SafeLOGIC*)
	visuAcknExtData : DownloadAcknExtMaOpTypeV1; (*acknowledge extended machine options*)
	visuAcknMachineOptions : ARRAY[0..511] OF BOOL; (*acknowledge machine options*)
	visuApplicationCRC : STRING[8]; (*CRC HEX string for visualization*)
	visuDeviceListInput : ARRAY[0..1] OF DownloadDeviceTypeV1; (*device list input*)
	visuDeviceListOutput : ARRAY[0..1] OF DownloadDeviceTypeV1; (*device list output*)
	visuDintInput : ConfigurationDintOptionsTypeV1; (*DINT channels input*)
	visuDintOutput : ConfigurationDintOptionsTypeV1; (*DINT channels output*)
	visuEnableDINTOptions : BOOL; (*enable DINT options*)
	visuEnableINTOptions : BOOL; (*enable INT options*)
	visuEnableMachineOptions : BOOL; (*enable BIT options*)
	visuEnableModuleFlags : BOOL; (*enable module flags*)
	visuEnableUDINTOptions : BOOL; (*enable UDINT options*)
	visuEnableUINTOptions : BOOL; (*enable UINT options*)
	visuIntInput : ConfigurationIntOptionsTypeV1; (*INT channels input*)
	visuIntOutput : ConfigurationIntOptionsTypeV1; (*INT channels output*)
	visuMachineOptionsBitInput : ARRAY[0..511] OF BOOL; (*BIT options input*)
	visuMachineOptionsBitOutput : ARRAY[0..511] OF BOOL; (*BIT options output*)
	visuModuleFlagsNotPresentInput : ARRAY[0..1023] OF BOOL; (*not present module flags input*)
	visuModuleFlagsNotPresentOutput : ARRAY[0..1023] OF BOOL; (*not present module flags output*)
	visuModuleFlagsOptionalInput : ARRAY[0..1023] OF BOOL; (*optional module flags input*)
	visuModuleFlagsOptionalOutput : ARRAY[0..1023] OF BOOL; (*optional module flags output*)
	visuModuleFlagsStartupInput : ARRAY[0..1023] OF BOOL; (*startup module flags input*)
	visuModuleFlagsStartupOutput : ARRAY[0..1023] OF BOOL; (*startup module flags output*)
	visuUDID_High : STRING[8]; (*UDID hex string for visualization*)
	visuUDID_Low : STRING[8]; (*UDID hex string for visualization*)
	visuUdintInput : ConfigurationUdintOptionsTypeV1; (*UDINT channels input*)
	visuUdintOutput : ConfigurationUdintOptionsTypeV1; (*UDINT channels output*)
	visuUintInput : ConfigurationUintOptionsTypeV1; (*UINT channels input*)
	visuUintOutput : ConfigurationUintOptionsTypeV1; (*UINT channels output*)
	visuUsedSLIDData : UINT; (*SafeLOGIC ID for data download*)
	visuUsedSLIDRemote : UINT; (*SafeLOGIC ID for remote control*)
	xcnt : UINT; (*counter variable*)
END_VAR
```

#### SafetySample.fun - Useful functions
```iecst
(********************************************************************
 * COPYRIGHT -- Bernecker + Rainer
 ********************************************************************
 * Program: SafetySample
 * File: SafetySample.fun
 * Author: B&R
 ********************************************************************
 * Functions and function blocks of program SafetySample
 ********************************************************************)

FUNCTION itoahex : UINT (*converts a UDINT values into a HEX character string*) (*$GROUP=User*)
	VAR_INPUT
		value : UDINT; (*UDINT value to be converted into a HEX character string*)
		pString : UDINT; (*pointer to the destination character string*)
	END_VAR
	VAR
		i_counter : USINT; (*internal variable*)
		i_value : UDINT; (*internal variable*)
		i_cvalue : USINT; (*internal variable*)
	END_VAR
END_FUNCTION
```

#### itoahex.st - converts a UDINT values into a HEX character string
```iecst
(********************************************************************
 * COPYRIGHT -- Bernecker + Rainer
 ********************************************************************
 * Program: SafetySample
 * File: itoahex.st
 * Author: B&R
 ********************************************************************
 * Implementation of program SafetySample
 ********************************************************************)

(* converts a UDINT values into a HEX character string *)
FUNCTION itoahex

	i_value := value;

	FOR i_counter := 0 TO 7 BY 1  DO
		i_cvalue := REAL_TO_USINT(brmfloor(UDINT_TO_REAL(i_value / REAL_TO_UDINT(EXPT(16, 7 - i_counter)))));
		IF i_cvalue = 0 THEN
			brsmemset(pString + i_counter, 48, 1); // 48 Dec = ASCII '0'
		ELSIF i_cvalue > 0 AND i_cvalue < 10 THEN
			brsitoa(i_cvalue, pString + i_counter);
		ELSIF i_cvalue >= 10 THEN
			brsmemset(pString + i_counter, i_cvalue + 55, 1); // 65 Dec = ASCII 'A'
		END_IF

		IF i_cvalue > 0 THEN
			i_value := i_value - REAL_TO_UDINT(EXPT(16, 7 - i_counter)) * i_cvalue;
		END_IF

	END_FOR

	itoahex := 0;

END_FUNCTION
```

- Visualisation Logical/AsSafetySolution/Panel (not shown)

### Program Logical/alarm_management

#### Variables.var
```iecst
VAR
	MpAlarmXCore_0 : MpAlarmXCore;
	MpAlarmXListUI_0 : MpAlarmXListUI;
	MpAlarmXListUIConnect : MpAlarmXListUIConnectType;
END_VAR
```

#### Cyclic.st
```iecst
PROGRAM _CYCLIC

	MpAlarmXCore_0.MpLink := ADR(gAlarmXCore);
	MpAlarmXCore_0.Enable := 1;

	MpAlarmXCore_0();

	IF airPresureOK THEN
		MpAlarmXReset(gAlarmXCore,'AirPressureNotOK');
	ELSE
		MpAlarmXSet(gAlarmXCore,'AirPressureNotOK');
	END_IF

END_PROGRAM
```

### Program Logical/misc/misc (IEC)

#### Main.st
```iecst
PROGRAM _INIT

	doSafetyCurtainSupplyP11 := TRUE;
	doSafetyCurtainSupplyP15 := TRUE;
	doSafetyCurtainSupplyP17 := TRUE;

	doSignColumnGreen;
	doSignColumnOrange;
	doSignColumnRed;
	doSignColumnHorn;

END_PROGRAM

PROGRAM _CYCLIC

	sumEDM := BOOL_TO_INT(diMagazineEDM) + BOOL_TO_INT(diPalletizationEDM) + BOOL_TO_INT(diOutfeedEDM);

	CASE sumEDM OF
		0:
			MTBasicsPWM_0.DutyCycle := 100;
		1:
			MTBasicsPWM_0.DutyCycle := 50;
		2:
			MTBasicsPWM_0.DutyCycle := 50;
		3:
			MTBasicsPWM_0.DutyCycle := 0;
	END_CASE

	MTBasicsPWM_0(Enable := 1, Period := 1);

	doLedOn := MTBasicsPWM_0.Out;

	doLedOff := NOT doLedOn;

	diActivateAllSafetyCircuits;

	//signalization column
	doSignColumnRed := doLedOff;

	sumAuto := BOOL_TO_INT(modeZoneMagazine = modeZoneAuto) + BOOL_TO_INT(modeZonePalletization = modeZoneAuto) + BOOL_TO_INT(modeZoneOutfeed = modeZoneAuto);

	CASE sumAuto OF
		0:
			MTBasicsPWM_1.DutyCycle := 0;
		1:
			MTBasicsPWM_1.DutyCycle := 50;
		2:
			MTBasicsPWM_1.DutyCycle := 50;
		3:
			MTBasicsPWM_1.DutyCycle := 100;
	END_CASE

	MTBasicsPWM_1(Enable := 1, Period := 1);

	doSignColumnGreen := MTBasicsPWM_1.Out;

	MTBasicsPWM_2(Enable := alarmPresent, DutyCycle := 50, Period := 1);

	doSignColumnOrange := MTBasicsPWM_2.Out OR bypassHorn;

	IF release THEN
		doSignColumnHorn := MTBasicsPWM_2.Out AND NOT bypassHorn;
	END_IF

	IF NOT alarmPresent THEN
		bypassHorn := FALSE;
	END_IF

	IF alarmPresent AND diReset THEN
		bypassHorn := TRUE;
	END_IF

END_PROGRAM
```

### pallet_magazine.var
```iecst
VAR
	palletMagazineViolation : BOOL;
END_VAR
```

### Program Logical/pallett_magazine/pallet_magazine (IEC) - pallet magazine control

#### Main.st
```iecst
(*Control OF pallet magazine, also called "zásobník palet" nebo "stohovač" *)

PROGRAM _INIT

END_PROGRAM

PROGRAM _CYCLIC

	CASE modeOfOperation OF

		notReadyToStart: //the automat is not ready to start
			IF NOT palletMagazineViolation AND airPresureOK THEN
				modeOfOperation := readyToStart;
			END_IF

		readyToStart:

			IF cmdManualMode OR cmdAllToManualMode THEN
				modeOfOperation := manualMode;
			END_IF

		manualMode:

	END_CASE;

	//action to control the arms
	ArmsControl;

	palletDetected;

	(* error detection *)
	IF palletMagazineViolation THEN
		MpAlarmXSet(gAlarmXCore,'PalletMagazineViolation');
	ELSE
		MpAlarmXReset(gAlarmXCore,'PalletMagazineViolation');
	END_IF

END_PROGRAM
```

#### Types.typ - Local data types
```iecst
TYPE
	MagazineState :
		(
		undefinedState1,
		upperPosition,
		middlePosition,
		lowerPosition
		);
	ArmsState :
		(
		undefinedState,
		armsOpened,
		armsClosed
		);
	ModeOfOperation :
		(
		notReadyToStart,
		readyToStart,
		automatMode,
		manualMode,
		errorState
		);
END_TYPE
```

#### Variables.var - Local variables
```iecst
VAR
	cmdManualMode : BOOL; (*VISU:switches pallet magazine to manual mode*)
	modeOfOperation : ModeOfOperation;
	palletMagazineViolation : BOOL; (*safety violation*)
	closeArms : BOOL;
	openArms : BOOL;
	cmdCloseArms : BOOL; (*VISU:command to close the arms*)
	cmdOpenArms : BOOL; (*VISU:commad to open the arms*)
	armsState : ArmsState; (*VISU:arms state*)
	leftArmOpened : BOOL;
	leftArmClosed : BOOL;
	rightArmOpened : BOOL;
	rightArmClosed : BOOL;
	palletDetected : BOOL; (*pallet detected on conveyor P12*)
	TON_CloseLeftRequest : TON;
	TON_CloseRightRequest : TON;
	TON_OpenLeftRequest : TON;
	TON_OpenRightRequest : TON;
END_VAR
```

#### arms.st
```iecst
(* control of arms *)

ACTION ArmsControl:

	// get arms state
	armsState := undefinedState;

	IF leftArmClosed AND rightArmClosed AND NOT leftArmOpened AND NOT rightArmOpened THEN
		armsState := armsClosed;
	END_IF

	IF leftArmOpened AND rightArmOpened AND NOT leftArmClosed AND NOT rightArmClosed THEN
		armsState := armsOpened;
	END_IF

	// command to close
	IF cmdCloseArms THEN
		//set output
		closeArms := TRUE;
		(* invert second output *)
		openArms := NOT closeArms;
	END_IF

	// command to open
	IF cmdOpenArms THEN
		//set output
		closeArms := FALSE;
		(* invert second output *)
		openArms := NOT closeArms;
	END_IF

	//close left check
	TON_CloseLeftRequest.IN := closeArms;
	TON_CloseLeftRequest.PT := T#6s;
	IF leftArmClosed THEN
		TON_CloseLeftRequest.IN := FALSE;
	END_IF

	TON_CloseLeftRequest();

	IF TON_CloseLeftRequest.Q THEN
		MpAlarmXSet(gAlarmXCore,'LeftArmNotClosed');
	ELSE
		MpAlarmXReset(gAlarmXCore,'LeftArmNotClosed');
	END_IF

	//close right check
	TON_CloseRightRequest.IN := closeArms;
	TON_CloseRightRequest.PT := T#6s;
	IF rightArmClosed THEN
		TON_CloseRightRequest.IN := FALSE;
	END_IF

	TON_CloseRightRequest();

	IF TON_CloseRightRequest.Q THEN
		MpAlarmXSet(gAlarmXCore,'RightArmNotClosed');
	ELSE
		MpAlarmXReset(gAlarmXCore,'RightArmNotClosed');
	END_IF

	//open left check
	TON_OpenLeftRequest.IN := openArms;
	TON_OpenLeftRequest.PT := T#6s;
	IF leftArmOpened THEN
		TON_OpenLeftRequest.IN := FALSE;
	END_IF

	TON_OpenLeftRequest();

	IF TON_OpenLeftRequest.Q THEN
		MpAlarmXSet(gAlarmXCore,'LeftArmNotOpened');
	ELSE
		MpAlarmXReset(gAlarmXCore,'LeftArmNotOpened');
	END_IF

	//open right check
	TON_OpenRightRequest.IN := openArms;
	TON_OpenRightRequest.PT := T#6s;
	IF rightArmOpened THEN
		TON_OpenRightRequest.IN := FALSE;
	END_IF

	TON_OpenRightRequest();

	IF TON_OpenRightRequest.Q THEN
		MpAlarmXSet(gAlarmXCore,'RightArmNotOpened');
	ELSE
		MpAlarmXReset(gAlarmXCore,'RightArmNotOpened');
	END_IF

END_ACTION
```

#### Cyclic.st - not listed in the package file held
```iecst
(* Control of pallet magazine, also called "zásobník palet" nebo "stohovač" *)

PROGRAM _CYCLIC

	CASE modeOfOperation OF

		notReadyToStart: //the automat is not ready to start
			IF NOT PalletMagazineViolation AND airPresureOK THEN
				modeOfOperation := readyToStart;
			END_IF

		readyToStart:

			IF cmdManualMode OR cmdAllToManualMode THEN
				modeOfOperation := manualMode;
			END_IF

		manualMode:
			IF cmdCloseArms THEN
				closeArms := TRUE;
				openArms := FALSE;
			END_IF

			IF cmdOpenArms THEN
				closeArms := FALSE;
				openArms := TRUE;
			END_IF

	END_CASE;

	IF palletMagazineViolation THEN
		MpAlarmXSet(gAlarmXCore,'PalletMagazineViolation');
	ELSE
		MpAlarmXReset(gAlarmXCore,'PalletMagazineViolation');
	END_IF

END_PROGRAM
```

### safety.var
```iecst
VAR
	diActivateAllSafetyCircuits : BOOL; (*button on main cabinet to activate all safety circuits*)
	diMagazineEDM : BOOL; (*magazine safety zone: 0...contactor switched on*)
	diPalletizationEDM : BOOL; (*paletization safety zone: 0...contactor switched on*)
	diOutfeedEDM : BOOL; (*wrapper+outfeed safety zone: 0...contactor switched on*)
END_VAR
```

### Program Logical/safety/safety (IEC)

#### Variables.var
```iecst
VAR
	doLedOn : BOOL; (*LED indicator on main cabinet*)
	doLedOff : BOOL; (*LED indicator on main cabinet*)
	MTBasicsPWM_0 : MTBasicsPWM;
	sum : INT;
	doSafetyCurtainSupplyP15 : BOOL;
	doSafetyCurtainSupplyP17 : BOOL;
	doSafetyCurtainSupplyP11 : BOOL;
END_VAR
```

#### Cyclic.st
```iecst
PROGRAM _CYCLIC

	IF diEStop1 THEN
		MpAlarmXReset(gAlarmXCore,'EStop1');
	ELSE
		MpAlarmXSet(gAlarmXCore,'EStop1');
	END_IF

	IF diEStop2 THEN
		MpAlarmXReset(gAlarmXCore,'EStop2');
	ELSE
		MpAlarmXSet(gAlarmXCore,'EStop2');
	END_IF

	IF diEStop3 THEN
		MpAlarmXReset(gAlarmXCore,'EStop3');
	ELSE
		MpAlarmXSet(gAlarmXCore,'EStop3');
	END_IF

	IF diEStop4 THEN
		MpAlarmXReset(gAlarmXCore,'EStop4');
	ELSE
		MpAlarmXSet(gAlarmXCore,'EStop4');
	END_IF

	IF diEStop5 THEN
		MpAlarmXReset(gAlarmXCore,'EStop5');
	ELSE
		MpAlarmXSet(gAlarmXCore,'EStop5');
	END_IF

	IF diEStopRobot THEN
		MpAlarmXReset(gAlarmXCore,'EStopRobot');
	ELSE
		MpAlarmXSet(gAlarmXCore,'EStopRobot');
	END_IF

	IF diEStopWrapper THEN
		MpAlarmXReset(gAlarmXCore,'EStopWrapper');
	ELSE
		MpAlarmXSet(gAlarmXCore,'EStopWrapper');
	END_IF

END_PROGRAM
```

#### Main.st
```iecst
PROGRAM _INIT

	doSafetyCurtainSupplyP11 := TRUE;
	doSafetyCurtainSupplyP15 := TRUE;
	doSafetyCurtainSupplyP17 := TRUE;

END_PROGRAM

PROGRAM _CYCLIC

	sum := BOOL_TO_INT(diMagazineEDM) + BOOL_TO_INT(diPalletizationEDM) + BOOL_TO_INT(diOutfeedEDM);

	CASE sum OF
		0:
			MTBasicsPWM_0.DutyCycle := 100;
		1:
			MTBasicsPWM_0.DutyCycle := 50;
		2:
			MTBasicsPWM_0.DutyCycle := 50;
		3:
			MTBasicsPWM_0.DutyCycle := 0;
	END_CASE

	MTBasicsPWM_0(Enable := 1, Period := 1);

	doLedOn := MTBasicsPWM_0.Out;

	doLedOff := NOT doLedOn;

	diActivateAllSafetyCircuits;

END_PROGRAM
```

### Variables.var - not listed in the package file held
```iecst
VAR
	activateSafetyCircuit : BOOL;
END_VAR
```

Listed in the project but not available here: Logical/Global.typ, Logical/Libraries/AcpInoSdc/Types.typ, Logical/Libraries/AcpInoSdc/Constants.var, Logical/Libraries/Atrima/Constants.var, Logical/Libraries/Misc/Constants.var, Logical/plc/palletization/palletization_main/palletization_main.typ, Logical/plc/palletization/pallet_conveyors/pallet_conveyors/Types.typ, Logical/plc/outfeed/outfeed_main/outfeed_main.typ, Logical/plc/outfeed/pallet_outfeed/pallet_outfeed/Types.typ, Logical/plc/outfeed/pallet_outfeed/pallet_outfeed/conveyorP17.st, Logical/plc/product_infeed/product_infeed.var, Logical/plc/product_infeed/product_infeed/Types.typ, Logical/plc/product_infeed/product_infeed/Variables.var, Logical/plc/robot_control/robot_control.var, Logical/plc/wrapper/wrapper.var, Logical/misc/misc.var, Logical/pallett_magazine/pallet_magazine/magazine.st, Logical/pallett_magazine/Program
